(* Logix 5000 project; controller DispersionPlc vendor 1 type 14 code 108 rev 34.11; software revision 34.01; part 2 of 22 *)
(* tags used below, declared in another part *)
   TO_ALARM_MSG_DINT : DINT;

ADD_ON_INSTRUCTION AStd_VFD_AOI   (* revision 1.0 *)
VAR_IN_OUT
   VFD : AStd_VFD; {required}
END_VAR
VAR_INPUT
   Running_I : BOOL; {required}
   SpeedFdbk_I : REAL; {required}
   Disconnect_I : BOOL; {required}
   DriveFault_I : BOOL; {required}
END_VAR
VAR_OUTPUT
   Start_O : BOOL; {access Read Only, required}
   Stop_O : BOOL; {access Read Only, required}
   DirectionFWD_O : BOOL; {access Read Only, required}
   DirectionREV_O : BOOL; {required}
   SpeedCmd_O : REAL; {access Read Only, required}
   ClearFault_O : BOOL; {access Read Only, required}
   AutoS : BOOL; {access Read Only, visible}
   RunS : BOOL; {access Read Only, visible}
   ReverseS : BOOL; {access Read Only, visible}
   AlmS : BOOL; {access Read Only, visible}
END_VAR
VAR_INPUT
   cfgHasRunFdbk : BOOL := 1; {visible}
   cfgHasSpeedFdbk : BOOL := 1; {visible}
   cfgHasDISC : BOOL; {visible}
   cfgRawMin : REAL; {required}
   cfgRawMax : REAL := 32767.0; {required}
   cfgEUMin : REAL; {required}
   cfgEUMax : REAL := 100.0; {required}
END_VAR
VAR
   RuntimeHourTimer : TIMER := (PRE := 3600000); {access None}
END_VAR

ROUTINE Logic   (* ladder *)
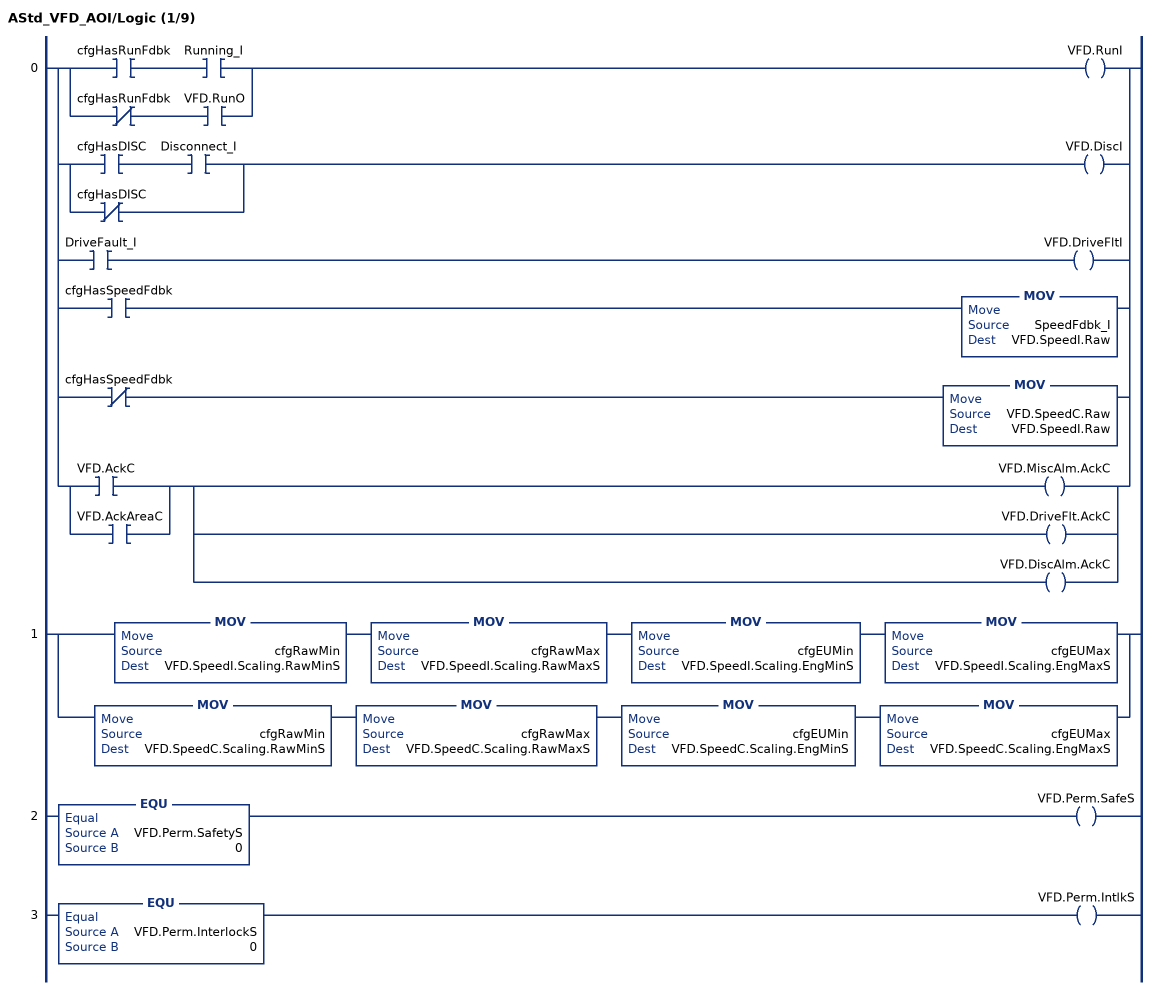
   0: [[XIC(cfgHasRunFdbk) XIC(Running_I) ,XIO(cfgHasRunFdbk) XIC(VFD.RunO) ] OTE(VFD.RunI) ,[XIC(cfgHasDISC) XIC(Disconnect_I) ,XIO(cfgHasDISC) ] OTE(VFD.DiscI) ,XIC(DriveFault_I) OTE(VFD.DriveFltI) ,[XIC(cfgHasSpeedFdbk) MOV(SpeedFdbk_I,VFD.SpeedI.Raw) ,XIO(cfgHasSpeedFdbk) MOV(VFD.SpeedC.Raw,VFD.SpeedI.Raw) ] ,[XIC(VFD.AckC) ,XIC(VFD.AckAreaC) ] [OTE(VFD.MiscAlm.AckC) ,OTE(VFD.DriveFlt.AckC) ,OTE(VFD.DiscAlm.AckC) ] ];
   1: [MOV(cfgRawMin,VFD.SpeedI.Scaling.RawMinS) MOV(cfgRawMax,VFD.SpeedI.Scaling.RawMaxS) MOV(cfgEUMin,VFD.SpeedI.Scaling.EngMinS) MOV(cfgEUMax,VFD.SpeedI.Scaling.EngMaxS) ,MOV(cfgRawMin,VFD.SpeedC.Scaling.RawMinS) MOV(cfgRawMax,VFD.SpeedC.Scaling.RawMaxS) MOV(cfgEUMin,VFD.SpeedC.Scaling.EngMinS) MOV(cfgEUMax,VFD.SpeedC.Scaling.EngMaxS) ];
   2: EQU(VFD.Perm.SafetyS,0)OTE(VFD.Perm.SafeS);
   3: EQU(VFD.Perm.InterlockS,0)OTE(VFD.Perm.IntlkS);
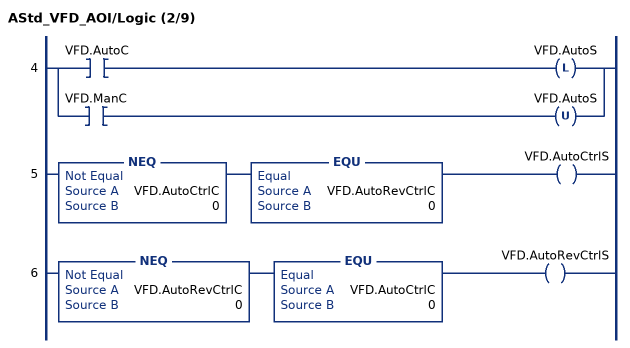
   4: [XIC(VFD.AutoC) OTL(VFD.AutoS) ,XIC(VFD.ManC) OTU(VFD.AutoS) ];
   5: NEQ(VFD.AutoCtrlC,0)EQU(VFD.AutoRevCtrlC,0)OTE(VFD.AutoCtrlS);
   6: NEQ(VFD.AutoRevCtrlC,0)EQU(VFD.AutoCtrlC,0)OTE(VFD.AutoRevCtrlS);
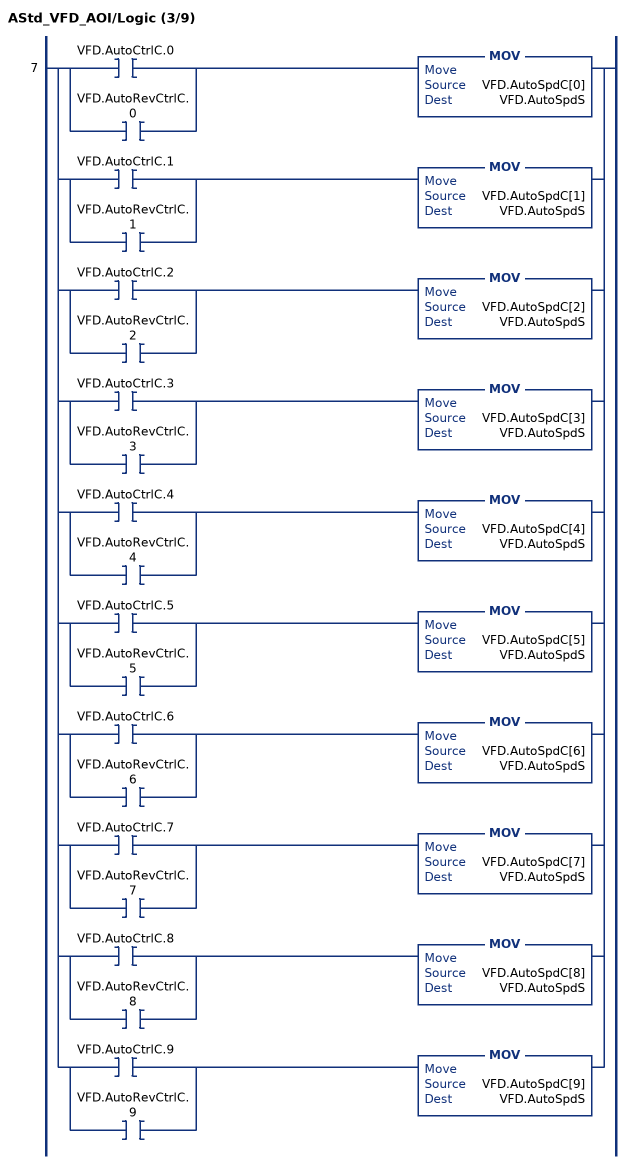
   7: [[XIC(VFD.AutoCtrlC.0) ,XIC(VFD.AutoRevCtrlC.0) ] MOV(VFD.AutoSpdC[0],VFD.AutoSpdS) ,[XIC(VFD.AutoCtrlC.1) ,XIC(VFD.AutoRevCtrlC.1) ] MOV(VFD.AutoSpdC[1],VFD.AutoSpdS) ,[XIC(VFD.AutoCtrlC.2) ,XIC(VFD.AutoRevCtrlC.2) ] MOV(VFD.AutoSpdC[2],VFD.AutoSpdS) ,[XIC(VFD.AutoCtrlC.3) ,XIC(VFD.AutoRevCtrlC.3) ] MOV(VFD.AutoSpdC[3],VFD.AutoSpdS) ,[XIC(VFD.AutoCtrlC.4) ,XIC(VFD.AutoRevCtrlC.4) ] MOV(VFD.AutoSpdC[4],VFD.AutoSpdS) ,[XIC(VFD.AutoCtrlC.5) ,XIC(VFD.AutoRevCtrlC.5) ] MOV(VFD.AutoSpdC[5],VFD.AutoSpdS) ,[XIC(VFD.AutoCtrlC.6) ,XIC(VFD.AutoRevCtrlC.6) ] MOV(VFD.AutoSpdC[6],VFD.AutoSpdS) ,[XIC(VFD.AutoCtrlC.7) ,XIC(VFD.AutoRevCtrlC.7) ] MOV(VFD.AutoSpdC[7],VFD.AutoSpdS) ,[XIC(VFD.AutoCtrlC.8) ,XIC(VFD.AutoRevCtrlC.8) ] MOV(VFD.AutoSpdC[8],VFD.AutoSpdS) ,[XIC(VFD.AutoCtrlC.9) ,XIC(VFD.AutoRevCtrlC.9) ] MOV(VFD.AutoSpdC[9],VFD.AutoSpdS) ];
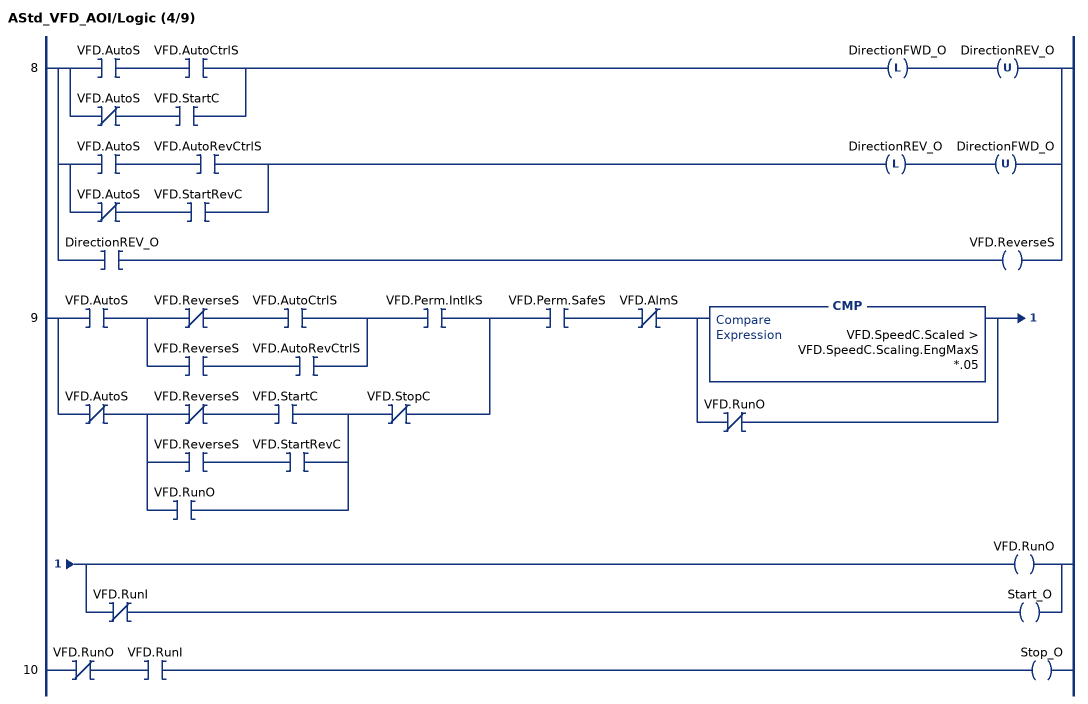
   8: [[XIC(VFD.AutoS) XIC(VFD.AutoCtrlS) ,XIO(VFD.AutoS) XIC(VFD.StartC) ] OTL(DirectionFWD_O) OTU(DirectionREV_O) ,[XIC(VFD.AutoS) XIC(VFD.AutoRevCtrlS) ,XIO(VFD.AutoS) XIC(VFD.StartRevC) ] OTL(DirectionREV_O) OTU(DirectionFWD_O) ,XIC(DirectionREV_O) OTE(VFD.ReverseS) ];
   9: [XIC(VFD.AutoS) [XIO(VFD.ReverseS) XIC(VFD.AutoCtrlS) ,XIC(VFD.ReverseS) XIC(VFD.AutoRevCtrlS) ] XIC(VFD.Perm.IntlkS) ,XIO(VFD.AutoS) [XIO(VFD.ReverseS) XIC(VFD.StartC) ,XIC(VFD.ReverseS) XIC(VFD.StartRevC) ,XIC(VFD.RunO) ] XIO(VFD.StopC) ]XIC(VFD.Perm.SafeS)XIO(VFD.AlmS)[CMP(VFD.SpeedC.Scaled > VFD.SpeedC.Scaling.EngMaxS *.05) ,XIO(VFD.RunO) ][OTE(VFD.RunO) ,XIO(VFD.RunI) OTE(Start_O) ];
   10: XIO(VFD.RunO)XIC(VFD.RunI)OTE(Stop_O);
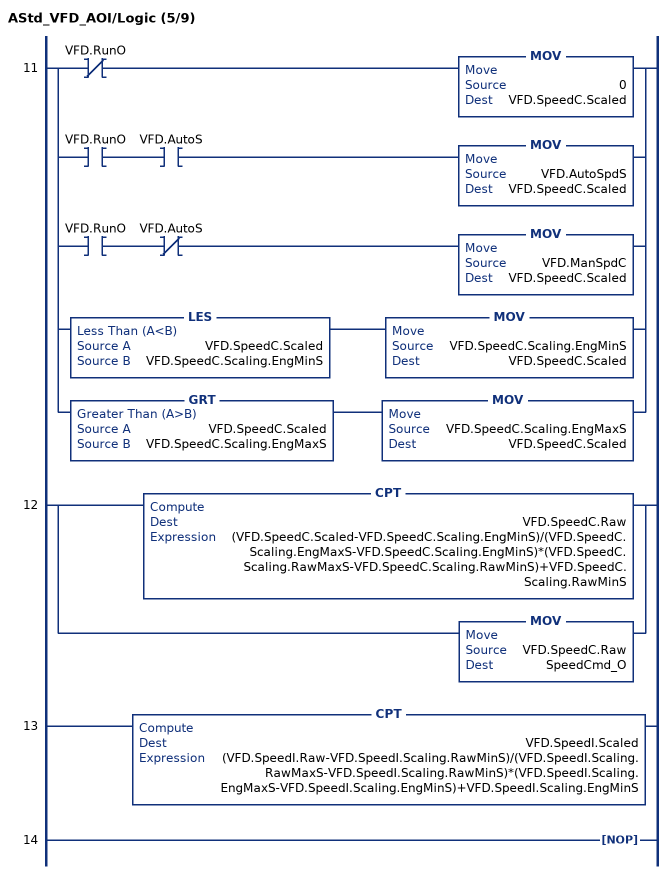
   11: [XIO(VFD.RunO) MOV(0,VFD.SpeedC.Scaled) ,XIC(VFD.RunO) XIC(VFD.AutoS) MOV(VFD.AutoSpdS,VFD.SpeedC.Scaled) ,XIC(VFD.RunO) XIO(VFD.AutoS) MOV(VFD.ManSpdC,VFD.SpeedC.Scaled) ,LES(VFD.SpeedC.Scaled,VFD.SpeedC.Scaling.EngMinS) MOV(VFD.SpeedC.Scaling.EngMinS,VFD.SpeedC.Scaled) ,GRT(VFD.SpeedC.Scaled,VFD.SpeedC.Scaling.EngMaxS) MOV(VFD.SpeedC.Scaling.EngMaxS,VFD.SpeedC.Scaled) ];
   12: [CPT(VFD.SpeedC.Raw,(VFD.SpeedC.Scaled-VFD.SpeedC.Scaling.EngMinS)/(VFD.SpeedC.Scaling.EngMaxS-VFD.SpeedC.Scaling.EngMinS)*(VFD.SpeedC.Scaling.RawMaxS-VFD.SpeedC.Scaling.RawMinS)+VFD.SpeedC.Scaling.RawMinS) ,MOV(VFD.SpeedC.Raw,SpeedCmd_O) ];
   13: CPT(VFD.SpeedI.Scaled,(VFD.SpeedI.Raw-VFD.SpeedI.Scaling.RawMinS)/(VFD.SpeedI.Scaling.RawMaxS-VFD.SpeedI.Scaling.RawMinS)*(VFD.SpeedI.Scaling.EngMaxS-VFD.SpeedI.Scaling.EngMinS)+VFD.SpeedI.Scaling.EngMinS);
   14: NOP();
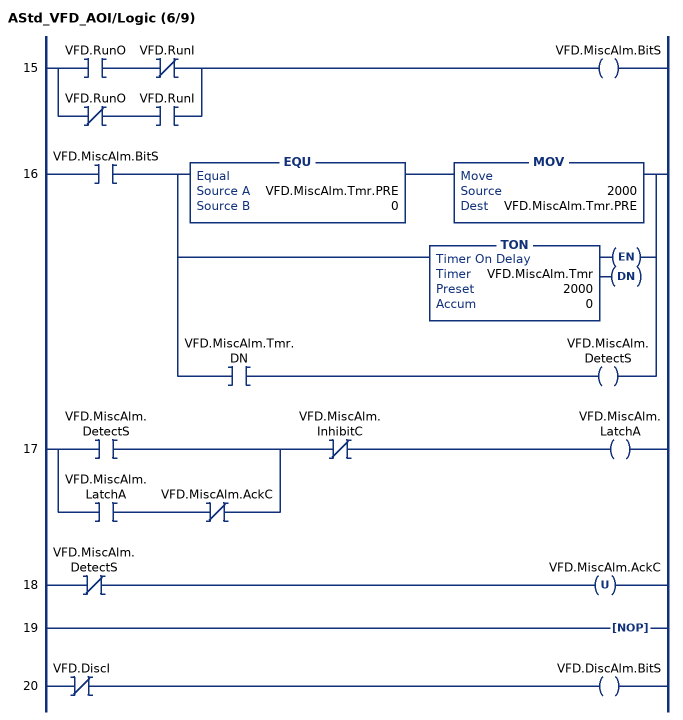
   15: [XIC(VFD.RunO) XIO(VFD.RunI) ,XIO(VFD.RunO) XIC(VFD.RunI) ]OTE(VFD.MiscAlm.BitS);
   16: XIC(VFD.MiscAlm.BitS)[EQU(VFD.MiscAlm.Tmr.PRE,0) MOV(2000,VFD.MiscAlm.Tmr.PRE) ,TON(VFD.MiscAlm.Tmr,2000,0) ,XIC(VFD.MiscAlm.Tmr.DN) OTE(VFD.MiscAlm.DetectS) ];
   17: [XIC(VFD.MiscAlm.DetectS) ,XIC(VFD.MiscAlm.LatchA) XIO(VFD.MiscAlm.AckC) ]XIO(VFD.MiscAlm.InhibitC)OTE(VFD.MiscAlm.LatchA);
   18: XIO(VFD.MiscAlm.DetectS)OTU(VFD.MiscAlm.AckC);
   19: NOP();
   20: XIO(VFD.DiscI)OTE(VFD.DiscAlm.BitS);
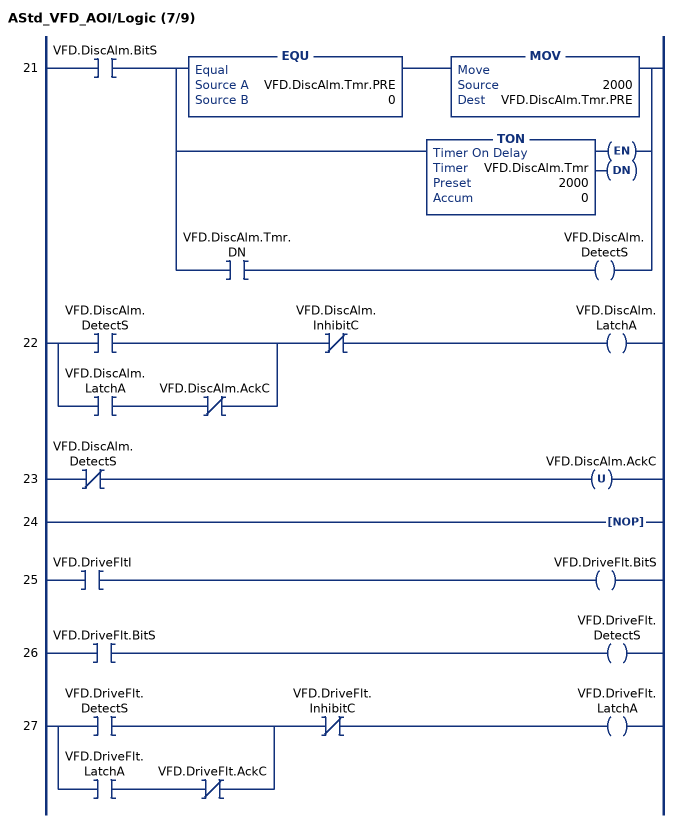
   21: XIC(VFD.DiscAlm.BitS)[EQU(VFD.DiscAlm.Tmr.PRE,0) MOV(2000,VFD.DiscAlm.Tmr.PRE) ,TON(VFD.DiscAlm.Tmr,2000,0) ,XIC(VFD.DiscAlm.Tmr.DN) OTE(VFD.DiscAlm.DetectS) ];
   22: [XIC(VFD.DiscAlm.DetectS) ,XIC(VFD.DiscAlm.LatchA) XIO(VFD.DiscAlm.AckC) ]XIO(VFD.DiscAlm.InhibitC)OTE(VFD.DiscAlm.LatchA);
   23: XIO(VFD.DiscAlm.DetectS)OTU(VFD.DiscAlm.AckC);
   24: NOP();
   25: XIC(VFD.DriveFltI)OTE(VFD.DriveFlt.BitS);
   26: XIC(VFD.DriveFlt.BitS)OTE(VFD.DriveFlt.DetectS);
   27: [XIC(VFD.DriveFlt.DetectS) ,XIC(VFD.DriveFlt.LatchA) XIO(VFD.DriveFlt.AckC) ]XIO(VFD.DriveFlt.InhibitC)OTE(VFD.DriveFlt.LatchA);
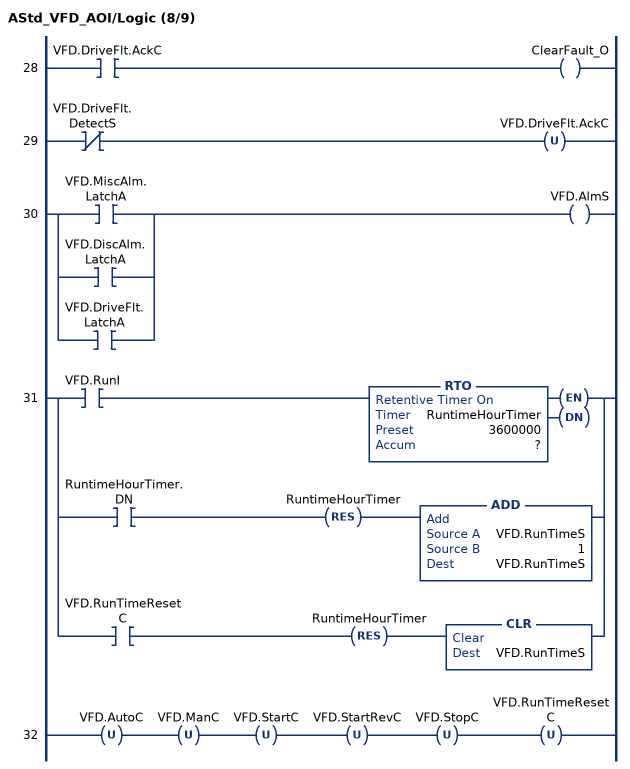
   28: XIC(VFD.DriveFlt.AckC)OTE(ClearFault_O);
   29: XIO(VFD.DriveFlt.DetectS)OTU(VFD.DriveFlt.AckC);
   30: [XIC(VFD.MiscAlm.LatchA) ,XIC(VFD.DiscAlm.LatchA) ,XIC(VFD.DriveFlt.LatchA) ]OTE(VFD.AlmS);
   31: [XIC(VFD.RunI) RTO(RuntimeHourTimer,?,?) ,XIC(RuntimeHourTimer.DN) RES(RuntimeHourTimer) ADD(VFD.RunTimeS,1,VFD.RunTimeS) ,XIC(VFD.RunTimeResetC) RES(RuntimeHourTimer) CLR(VFD.RunTimeS) ];
   32: OTU(VFD.AutoC)OTU(VFD.ManC)OTU(VFD.StartC)OTU(VFD.StartRevC)OTU(VFD.StopC)OTU(VFD.RunTimeResetC);
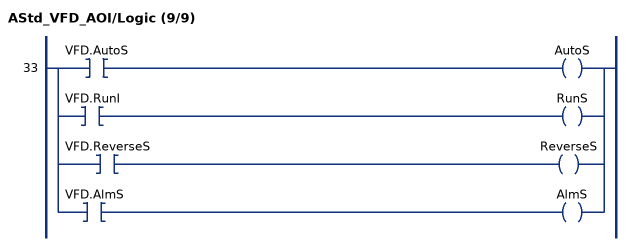
   33: [XIC(VFD.AutoS) OTE(AutoS) ,XIC(VFD.RunI) OTE(RunS) ,XIC(VFD.ReverseS) OTE(ReverseS) ,XIC(VFD.AlmS) OTE(AlmS) ];
END_ROUTINE
END_ADD_ON_INSTRUCTION

ADD_ON_INSTRUCTION AStd_VlVModulating_AOI   (* revision 1.0, vendor Avanceon *)
VAR_IN_OUT
   Valve : AStd_VlvModulating; {required}
END_VAR
VAR_INPUT
   cfgEUMin : REAL; {required}
   cfgEUMax : REAL := 100.0; {required}
   cfgRawMin : REAL := 4000.0; {required}
   cfgRawMax : REAL := 20000.0; {required}
END_VAR
VAR_OUTPUT
   OutputRaw_O : REAL; {required}
   AutoS : BOOL; {access Read Only, visible}
   OpenS : BOOL; {access Read Only, visible}
END_VAR
VAR
   ValveOpenRequest : BOOL; {access None}
END_VAR

ROUTINE Logic   (* ladder *)
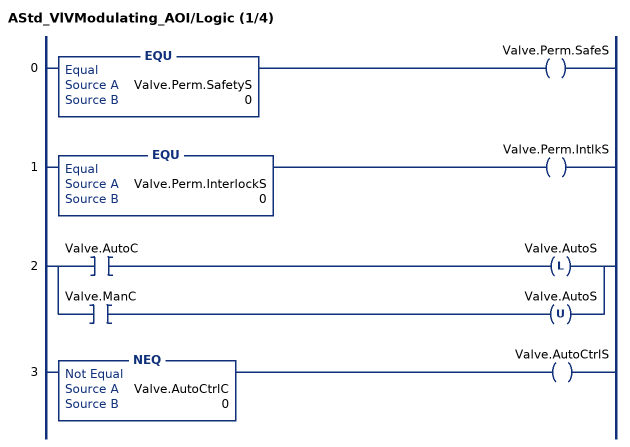
   0: EQU(Valve.Perm.SafetyS,0)OTE(Valve.Perm.SafeS);
   1: EQU(Valve.Perm.InterlockS,0)OTE(Valve.Perm.IntlkS);
   2: [XIC(Valve.AutoC) OTL(Valve.AutoS) ,XIC(Valve.ManC) OTU(Valve.AutoS) ];
   3: NEQ(Valve.AutoCtrlC,0)OTE(Valve.AutoCtrlS);
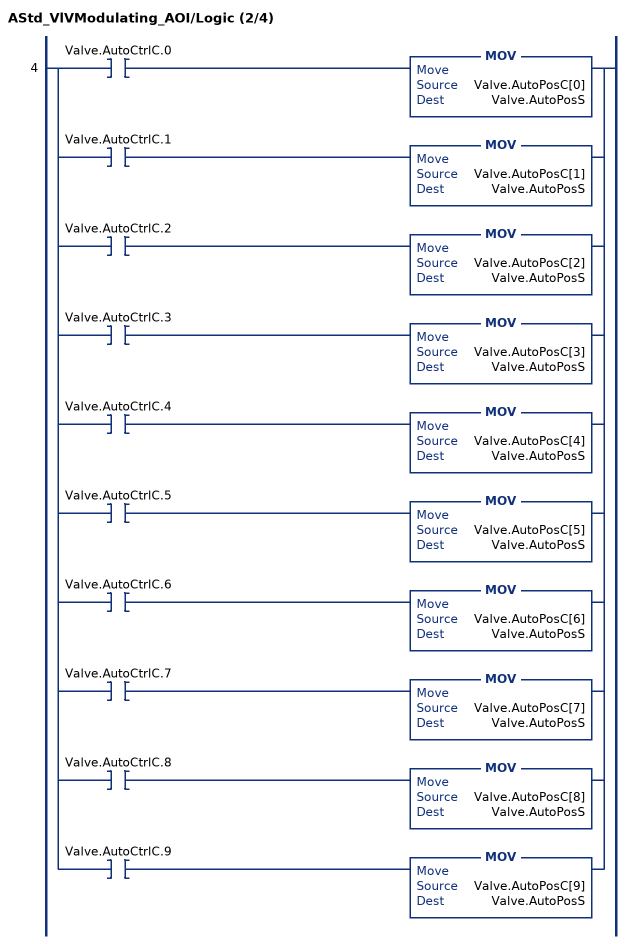
   4: [XIC(Valve.AutoCtrlC.0) MOV(Valve.AutoPosC[0],Valve.AutoPosS) ,XIC(Valve.AutoCtrlC.1) MOV(Valve.AutoPosC[1],Valve.AutoPosS) ,XIC(Valve.AutoCtrlC.2) MOV(Valve.AutoPosC[2],Valve.AutoPosS) ,XIC(Valve.AutoCtrlC.3) MOV(Valve.AutoPosC[3],Valve.AutoPosS) ,XIC(Valve.AutoCtrlC.4) MOV(Valve.AutoPosC[4],Valve.AutoPosS) ,XIC(Valve.AutoCtrlC.5) MOV(Valve.AutoPosC[5],Valve.AutoPosS) ,XIC(Valve.AutoCtrlC.6) MOV(Valve.AutoPosC[6],Valve.AutoPosS) ,XIC(Valve.AutoCtrlC.7) MOV(Valve.AutoPosC[7],Valve.AutoPosS) ,XIC(Valve.AutoCtrlC.8) MOV(Valve.AutoPosC[8],Valve.AutoPosS) ,XIC(Valve.AutoCtrlC.9) MOV(Valve.AutoPosC[9],Valve.AutoPosS) ];
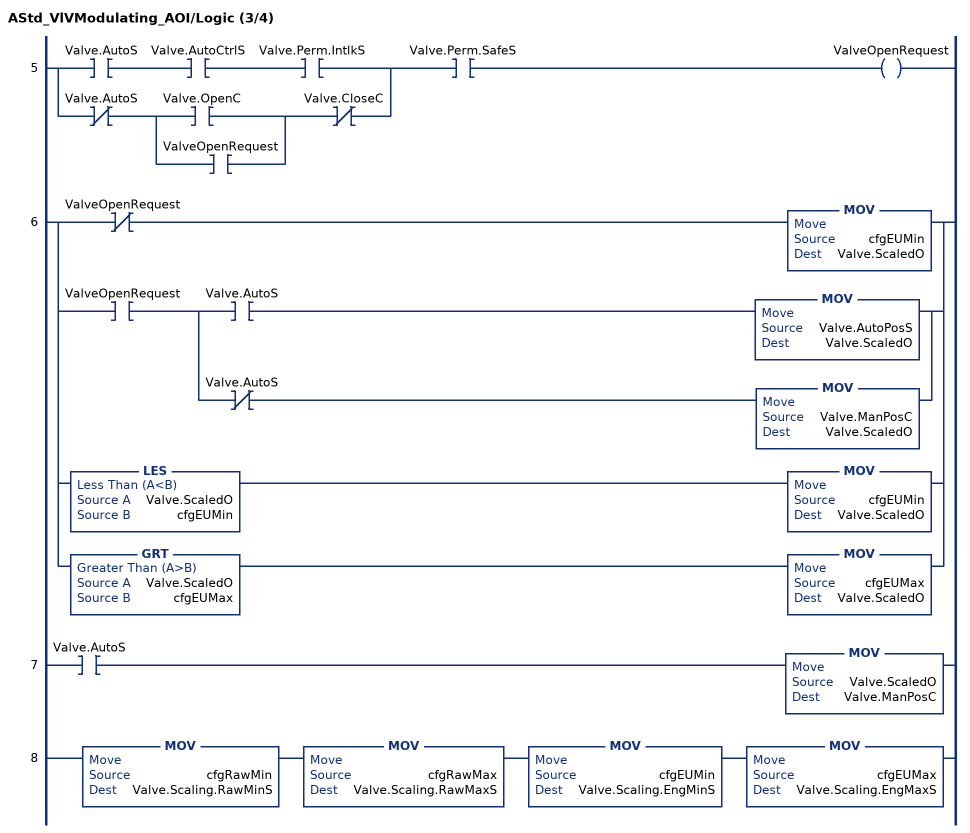
   5: [XIC(Valve.AutoS) XIC(Valve.AutoCtrlS) XIC(Valve.Perm.IntlkS) ,XIO(Valve.AutoS) [XIC(Valve.OpenC) ,XIC(ValveOpenRequest) ] XIO(Valve.CloseC) ]XIC(Valve.Perm.SafeS)OTE(ValveOpenRequest);
   6: [XIO(ValveOpenRequest) MOV(cfgEUMin,Valve.ScaledO) ,XIC(ValveOpenRequest) [XIC(Valve.AutoS) MOV(Valve.AutoPosS,Valve.ScaledO) ,XIO(Valve.AutoS) MOV(Valve.ManPosC,Valve.ScaledO) ] ,LES(Valve.ScaledO,cfgEUMin) MOV(cfgEUMin,Valve.ScaledO) ,GRT(Valve.ScaledO,cfgEUMax) MOV(cfgEUMax,Valve.ScaledO) ];
   7: XIC(Valve.AutoS)MOV(Valve.ScaledO,Valve.ManPosC);
   8: MOV(cfgRawMin,Valve.Scaling.RawMinS)MOV(cfgRawMax,Valve.Scaling.RawMaxS)MOV(cfgEUMin,Valve.Scaling.EngMinS)MOV(cfgEUMax,Valve.Scaling.EngMaxS);
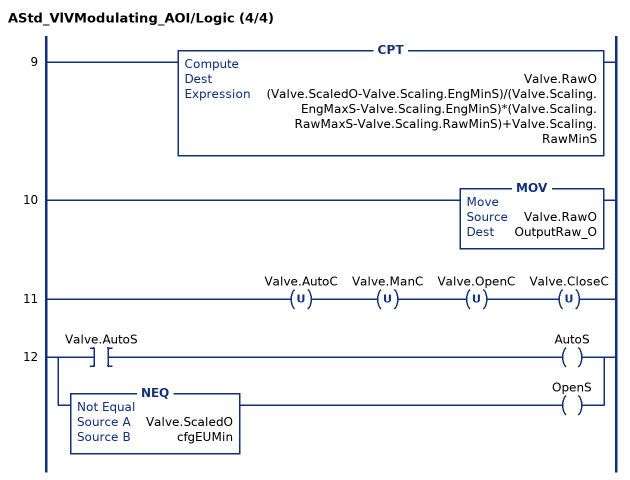
   9: CPT(Valve.RawO,(Valve.ScaledO-Valve.Scaling.EngMinS)/(Valve.Scaling.EngMaxS-Valve.Scaling.EngMinS)*(Valve.Scaling.RawMaxS-Valve.Scaling.RawMinS)+Valve.Scaling.RawMinS);
   10: MOV(Valve.RawO,OutputRaw_O);
   11: OTU(Valve.AutoC)OTU(Valve.ManC)OTU(Valve.OpenC)OTU(Valve.CloseC);
   12: [XIC(Valve.AutoS) OTE(AutoS) ,NEQ(Valve.ScaledO,cfgEUMin) OTE(OpenS) ];
END_ROUTINE
END_ADD_ON_INSTRUCTION

ADD_ON_INSTRUCTION AStd_VlvOC_AOI   (* revision 1.0, vendor Avanceon *)
VAR_IN_OUT
   Valve : AStd_VlvOC; {required}
END_VAR
VAR_OUTPUT
   AutoS : BOOL; {access Read Only, visible}
   OpenS : BOOL; {access Read Only, visible}
   AlmS : BOOL; {access Read Only, visible}
END_VAR
VAR_INPUT
   Open_I : BOOL; {required}
   Closed_I : BOOL; {required}
END_VAR
VAR_OUTPUT
   Open_O : BOOL; {required}
   Close_O : BOOL; {required}
END_VAR
VAR_INPUT
   cfgFailOpen : BOOL; {access None, visible}
   cfgHasZSO : BOOL := 1; {access None, visible}
   cfgHasZSC : BOOL; {access None, visible}
END_VAR
VAR
   ONS : SINT; {access None}
END_VAR

ROUTINE Logic   (* ladder *)
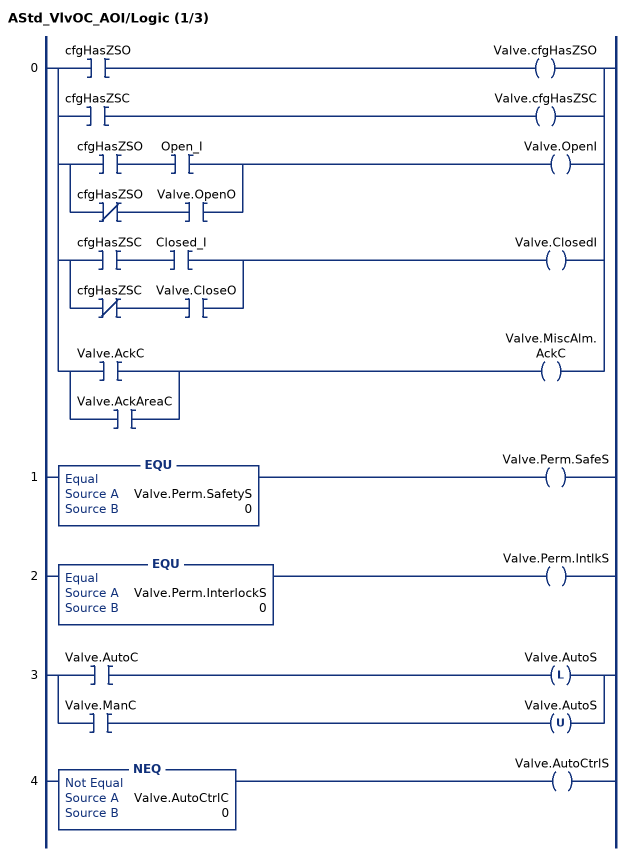
   0: [XIC(cfgHasZSO) OTE(Valve.cfgHasZSO) ,XIC(cfgHasZSC) OTE(Valve.cfgHasZSC) ,[XIC(cfgHasZSO) XIC(Open_I) ,XIO(cfgHasZSO) XIC(Valve.OpenO) ] OTE(Valve.OpenI) ,[XIC(cfgHasZSC) XIC(Closed_I) ,XIO(cfgHasZSC) XIC(Valve.CloseO) ] OTE(Valve.ClosedI) ,[XIC(Valve.AckC) ,XIC(Valve.AckAreaC) ] OTE(Valve.MiscAlm.AckC) ];
   1: EQU(Valve.Perm.SafetyS,0)OTE(Valve.Perm.SafeS);
   2: EQU(Valve.Perm.InterlockS,0)OTE(Valve.Perm.IntlkS);
   3: [XIC(Valve.AutoC) OTL(Valve.AutoS) ,XIC(Valve.ManC) OTU(Valve.AutoS) ];
   4: NEQ(Valve.AutoCtrlC,0)OTE(Valve.AutoCtrlS);
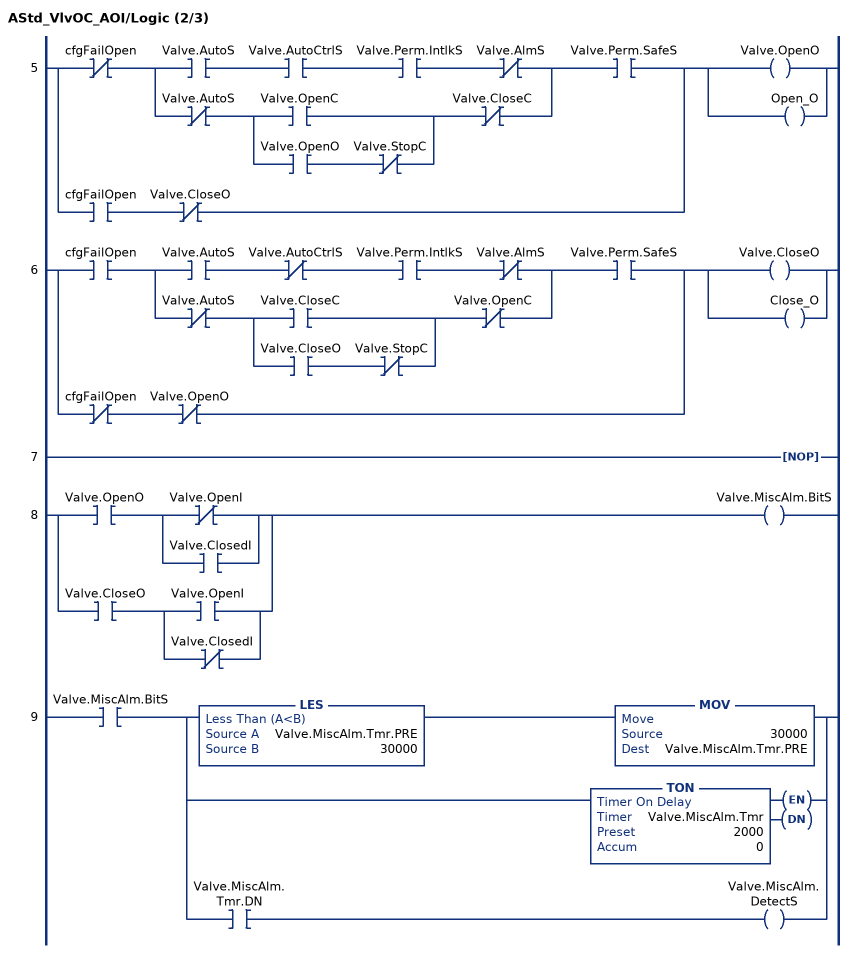
   5: [XIO(cfgFailOpen) [XIC(Valve.AutoS) XIC(Valve.AutoCtrlS) XIC(Valve.Perm.IntlkS) XIO(Valve.AlmS) ,XIO(Valve.AutoS) [XIC(Valve.OpenC) ,XIC(Valve.OpenO) XIO(Valve.StopC) ] XIO(Valve.CloseC) ] XIC(Valve.Perm.SafeS) ,XIC(cfgFailOpen) XIO(Valve.CloseO) ][OTE(Valve.OpenO) ,OTE(Open_O) ];
   6: [XIC(cfgFailOpen) [XIC(Valve.AutoS) XIO(Valve.AutoCtrlS) XIC(Valve.Perm.IntlkS) XIO(Valve.AlmS) ,XIO(Valve.AutoS) [XIC(Valve.CloseC) ,XIC(Valve.CloseO) XIO(Valve.StopC) ] XIO(Valve.OpenC) ] XIC(Valve.Perm.SafeS) ,XIO(cfgFailOpen) XIO(Valve.OpenO) ][OTE(Valve.CloseO) ,OTE(Close_O) ];
   7: NOP();
   8: [XIC(Valve.OpenO) [XIO(Valve.OpenI) ,XIC(Valve.ClosedI) ] ,XIC(Valve.CloseO) [XIC(Valve.OpenI) ,XIO(Valve.ClosedI) ] ]OTE(Valve.MiscAlm.BitS);
   9: XIC(Valve.MiscAlm.BitS)[LES(Valve.MiscAlm.Tmr.PRE,30000) MOV(30000,Valve.MiscAlm.Tmr.PRE) ,TON(Valve.MiscAlm.Tmr,2000,0) ,XIC(Valve.MiscAlm.Tmr.DN) OTE(Valve.MiscAlm.DetectS) ];
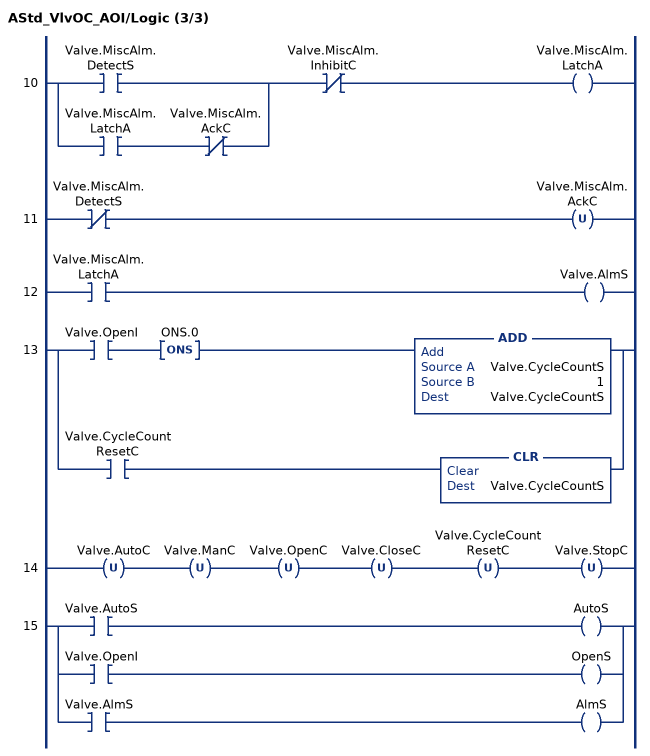
   10: [XIC(Valve.MiscAlm.DetectS) ,XIC(Valve.MiscAlm.LatchA) XIO(Valve.MiscAlm.AckC) ]XIO(Valve.MiscAlm.InhibitC)OTE(Valve.MiscAlm.LatchA);
   11: XIO(Valve.MiscAlm.DetectS)OTU(Valve.MiscAlm.AckC);
   12: XIC(Valve.MiscAlm.LatchA)OTE(Valve.AlmS);
   13: [XIC(Valve.OpenI) ONS(ONS.0) ADD(Valve.CycleCountS,1,Valve.CycleCountS) ,XIC(Valve.CycleCountResetC) CLR(Valve.CycleCountS) ];
   14: OTU(Valve.AutoC)OTU(Valve.ManC)OTU(Valve.OpenC)OTU(Valve.CloseC)OTU(Valve.CycleCountResetC)OTU(Valve.StopC);
   15: [XIC(Valve.AutoS) OTE(AutoS) ,XIC(Valve.OpenI) OTE(OpenS) ,XIC(Valve.AlmS) OTE(AlmS) ];
END_ROUTINE
END_ADD_ON_INSTRUCTION

VAR_GLOBAL   (* controller tags *)
   _bottom : REAL;
   _JISdebug : DINT := 2;
        .0   // Remapping
        .2   // Delete when probe is working
   _Placeholder : DINT := 1081857;
   _Placeholder_LS_4302_AI : REAL := 8.0;
   AFB : BOOL;
   AFI : BOOL;
   AG4302_LLP_Alarm : BOOL;
   AG4302_LLPower : TIMER := (PRE := 5000);
   AirMakeup : TIMER := (PRE := 2000);
   AirMakeup_BEAC : ALIAS FOR Local:1:O.Data[12].11;
   AirMakeup_BEACA : ALIAS FOR Local:1:O.Data[22].11;
   AMMONIUM_START_ATTEMP : BOOL;
   B4320_Amount_Per_Count : REAL;
   B4320_Charge_Remaining : REAL;
   B4320_Flow_Rate : REAL;
   B4320_Flow_Raw : DINT;
   B4320_Flow_Raw_Adjusted : REAL;
   B4320_Flow_Scale_Factor : REAL;
   B4320_HighHighLevel : BOOL;
   B4320_HighHighLevelMessage : BOOL;
   B4320_HighLevel : BOOL := 1;
   B4320_Last_Charge : DINT;
   B4320_LastTrasferredLb : REAL := 43900.0;
   B4320_Manual_Start : BOOL;
   B4320_Max_Flow : REAL;
   B4320_OkToRun : BOOL;
   B4320_Pump_Manual_Run : BOOL;
   B4320_Pump_Off : BOOL;
   B4320_Pump_Run : BOOL;
   B4320_PumpAutoCommand : BOOL;
   B4320_PumpManCommand : BOOL;
   B4320_PumpManStart : AOI_Toggle := (QNot := 1);
   B4320_Selected : BOOL;
   B4320_SelectPB : BOOL;
   B4320_Tank_Max_Lbs : REAL;
   B4320_Toggle : AOI_Toggle := (QNot := 1);
   B4320_Transfer : BOOL;
   B4320_transfer_amount : REAL;
   B4320_TransferDone : BOOL;
   B4320_TransferLimit : REAL := 44600.0;
   B4320_transferLimitMessage : BOOL;
   B4320_TransferSetpoint : REAL := 44000.0;
   B4320_TransferStarted : BOOL;
   B4320_TransferStartPB : BOOL;
   B4320_TransferStopPB : BOOL;
   B4320PumpTmr : TIMER;
   B4320SelectPB : BOOL;
   BarcodeBypassAcitve : BOOL;
   BarcodeBypassAcitvePB : BOOL;
   BarcodeForEditString : STRING := '01A0026';
   BarcodeIndex : DINT := 7;
   BarcodeIndex_Hold : DINT := 7;
   BarCodeReadHeartbeat : INT := 9751;
   BarcodeScan0NotOKDelay : TIMER := (PRE := 250);
   BarcodeScan1NotOKDelay : TIMER := (PRE := 250);
   BarcodeScan2NotOKDelay : TIMER := (PRE := 250);
   BarcodeScanBypass : BOOL := 1;
   BarcodeScanNotOK : INT;
   BarcodeScanOK : INT;
   BarcodeScanRequest : BOOL[32];
   BarcodeScanRequestPB : INT;
   BarcodeScanSequence : INT;
   bb : BOOL;
   BBVV : BOOL;
   BL_4310_AUX : ALIAS FOR Local:1:I.Data[1].2;
   BL_4310_RUN : ALIAS FOR Local:1:O.Data[0].2;
   BLANK64 : Stp64;
   BlankStrg : STRING;
   block_bit1 : BOOL := 1;
   block_bit2 : BOOL;
   bogus : BOOL;
   bogus_bit : BOOL;
   Both_Running : BOOL := 1;
   Both_Running_Timer : TIMER := (PRE := 3000, ACC := 3001, EN := 1, DN := 1);
   BUFENCTU : COUNTER := (PRE := 10000, ACC := 106);
   Bulk_Tank_T52_Level_Lamp : ALIAS FOR Local:1:O.Data[12].3;
   Bulk_Tank_T52_Level_LampA : ALIAS FOR Local:1:O.Data[12].3;
   Bulk_Tank_T52_Level_LampB : ALIAS FOR Local:1:O.Data[22].3;
   Bulk_Tank_T53_Level_Lamp : ALIAS FOR Local:1:O.Data[12].4;
   Bulk_Tank_T53_Level_LampA : ALIAS FOR Local:1:O.Data[22].4;
   bypass_bit : BOOL := 1;
   Capture_Delay : TIMER := (PRE := 3000);
   Capture_Delay_1 : TIMER := (PRE := 3000);
   Capture_Destination : DINT := 1;
   Capture_Destination_1 : DINT := 1;
   Capture_ONS : BOOL;
   Capture_ONS1 : BOOL;
   Capture_ONS_2 : BOOL;
   Capture_ONS_3 : BOOL;
   Capture_Selected : BOOL := 1;
   Capture_Selected_1 : BOOL;
   Cat_Destination_K400 : BOOL := 1;
   Cat_Destination_K400_ONS : BOOL;
   Cat_Destination_K400_PB : BOOL;
   Cat_Destination_T4301 : BOOL;
   Cat_Destination_T4301_ONS : BOOL;
   Cat_Destination_T4301_PB : BOOL;
   Cat_Destination_T4302 : BOOL;
   Cat_Destination_T4302_ONS : BOOL;
   Cat_Destination_T4302_PB : BOOL;
   Cat_Isolation_T430X_Timer : TIMER;
   Cat_Isolation_Valve_Timer : TIMER := (PRE := 120000);
   Cat_Man_ONS : BOOL;
   Cat_Pump_manual : BOOL;
   Cat_Purge_Transfer_K400 : Seq64 := (Sq.Step[0] := 1);
   Cat_Purge_Transfer_T430X : Seq64 := (Sq.Step[0] := 1);
   Cat_Recirc_Transfer_K400 : Seq64 := (Val := 6, Sq.Step[6] := 1);
   Cat_Recirc_Transfer_T430X : Seq64 := (Val := 1, Sq.Step[0] := 1);
   Cat_Scale_Factor : REAL := 0.0018;
   cat_start_dispencse : BOOL := 1;
   Cat_Tank_Destination : DINT := 1;
   cat_target_weight_bypass : BOOL;
   Cat_Zero : REAL := 4.03636;
   Catalyst_Destination : DINT;
   catalyst_MaxFeedRate : REAL := 3.4;
   CATALYST_RESET : BOOL;
   CatalystTimers_11_HMI : REAL := 7.01;
   CATFLOW : TIMER := (PRE := 500);
   CE_4301 : REAL := 0.17498249;
   ce_4301_High : REAL := 5.0;
   ce_4301_Low : REAL := -3.0;
   ce_4301_Max : REAL;
   CE_4301_OffSet : REAL := 4000.0;
   CE_4301_Sf : REAL := 0.0049995;
   CE_4302 : REAL := 0.129987;
   ce_4302_High : REAL := 15.0;
   CE_4302_Low : REAL := -3.0;
   CE_4302_OffSet : REAL := 4000.0;
   CE_4302_Sf : REAL := 0.0049995;
   Circulation_Timer_Continue : BOOL;
   constant : REAL := 10.0;
   constant1 : DINT := 1;
   Control_Rm_tags : DINT;
   Cool_Setpoint_4301 : DINT := 85;
   Cool_Setpoint_4302 : DINT := 180;
   Cool_SP : REAL := 15.0;
   Cool_SP2 : REAL := 17.5;
   Cool_SP3 : REAL := 20.0;
   Cool_SP4 : REAL := 100.0;
   CountTmr : TIMER := (PRE := 200);
   CR : STRING := '$0D';
   CRADT : ALIAS FOR Local:5:O.Data.7;
   Current4302FQ : REAL := 53.641064;
   CurrentTrasferredLb : REAL;
   dan1 : DINT := 112;
   dan2 : REAL := 1200.0;
   dan3 : BOOL;
   dan4 : BOOL := 1;
   dan5 : BOOL;
   dan6 : BOOL;
   dan99 : BOOL;
   dantoggle1 : BOOL := 1;
   DATAFDUNLATCH : TIMER := (PRE := 2000);
   DATAUNCOUNT : COUNTER := (PRE := 20000, ACC := 2198);
   ddd : BOOL := 1;
   Debug : DINT := 3;
   Dev : REAL[10] := ([0] := 2.8410683, [1] := 3.3833313);
   DevAck : DINT;
   DevAlarms : DINT := 60;
   DeviationFactor : REAL := 0.03;
   DevTimer : TIMER[10] := ([0].PRE := 30000, [1].PRE := 30000);
   Disp_AlarmsResetting : BOOL;
   Disp_Alr_To_Sound_Horn : BOOL[128] := ([10] := 1, [13] := 1, [14] := 1, [19] := 1, [25] := 1, [27] := 1, [28] := 1, [38] := 1, [44] := 1, [46] := 1, [51] := 1, [54] := 1, [55] := 1, [66] := 1, [70] := 1, [71] := 1, [87] := 1, [88] := 1, [99] := 1, [111] := 1, [115] := 1, [121] := 1, [122] := 1);
   Disp_AlrResetIdx : DINT := 127;
   Disp_QuedAlarm : DINT := 108;
   DispAlarmResetBit : BOOL;
   Dispersion_from_Main : DINT := 1;
   Dispersion_from_Main2 : DINT := 8131435;
   Dispersion_from_Main2_DintToStringConv : STRING := '8131435';
   Dispersion_from_SIL2 : DINT := 1;
   Dispersion_from_SIL2_Analog : REAL[24] := ([0] := 86.51327, [1] := 66.32967, [2] := 90.0, [10] := 152.36926);
   Dispersion_to_Main : DINT := 1;
   Dispersion_to_Main2 : DINT;
   Dispersion_to_SIL2 : DINT := 32;
   Dispersion_to_SIL2_Analog : REAL[24] := ([0] := 90.0, [1] := 10.0, [2] := 45.0, [3] := 15901.0, [4] := 15801.0);
   Dispersion_to_SIL2_Analog_xxx : DINT;
   DispersionAlarmReset : BOOL;
   DispersionAlarms : BOOL[256] := ([2] := 1, [103] := 1, [108] := 1, [157] := 1, [159] := 1, [250] := 1);
   DispersionProductID : STRING[21] := ([0] := '8131428', [1] := '8131435', [2] := '8132028', [3] := '8211377', [4] := '8212241', [5] := 'IDLE', [6] := '7108441');
   DispersionProductID_BarcodeScan : STRING;
   DispersionProductID_ScanIndex : DINT := 8;
   DispersionProductID_ScanIndex_Storage : DINT;
   DispersionProductIDEntryStorage : STRING;
   DispersionProductIDKeyEntry : STRING := '7108441';
   DispersionProductIDKeyEntry1 : STRING;
   DispersionProductIDMatch : STRING;
   DPT_4301 : REAL;
   dpt_4301_High : REAL := 40000.0;
   DPT_4301_Holding : REAL := 3900.84;
   DPT_4301_OffSet : REAL := 4000.0;
   DPT_4301_Samples : DINT := 1000;
   DPT_4301_Sf : REAL := 3.41875;
   DPT_4302 : REAL;
   dpt_4302_High : REAL := 35000.0;
   DPT_4302_Holding : REAL := 3917.319;
   DPT_4302_OffSet : REAL := 4000.0;
   DPT_4302_Samples : DINT := 100;
   DPT_4302_Sf : REAL := 3.41875;
   DPT_4303 : REAL := 7949.331;
   DPT_4303_High : REAL := 16300.0;
   DPT_4303_Holding : REAL := 10860.054;
   DPT_4303_OffSet : REAL := 4000.0;
   DPT_4303_Samples : DINT := 100;
   DPT_4303_Sf : REAL := 1.02186;
   DPT_4303_Tare_Val : REAL;
   DPT_4320 : REAL := 33840.145;
   DPT_4320_FILL : REAL := 1489.0;
   DPT_4320_High : REAL := 48500.0;
   DPT_4320_Holding1 : REAL := 14397.525;
   DPT_4320_OffSet : REAL := 3904.0;
   DPT_4320_Raw : INT := 14392;
   DPT_4320_Sf : REAL := 3.083;
   DPT_4320_Sf_old : REAL := 3.466;
   DPT_4320rev1 : REAL;
   dpthighraw : REAL := 20837.0;
   dptlowraw : REAL := -32.0;
   Drum_Addition_K400 : Seq64 := (Sq.Step[0] := 1, AutoMode := 1);
   Drum_Addition_T430X : Seq64 := (Sq.Step[0] := 1);
   Drum_Addition_T430X_Timer : TIMER := (PRE := 30000);
   Drum_Addition_Timer : TIMER := (PRE := 120000);
   Drum_Transfer : BOOL;
   Drum_Transfer_Active : BOOL;
   Drum_Transfer_ONS : BOOL;
   Drum_Transfer_ONS_1 : BOOL;
   Dummy_Safety_1 : BOOL[32];
   DummyOutput : BOOL := 1; {access None}
   Emergency_Cool_4301 : BOOL;
   Emergency_Cool_4301_Reset : BOOL;
   Emergency_Cool_4302 : BOOL;
   Emergency_Cool_4302_Reset : BOOL;
   Enable_High_Alarm : BOOL := 1;
   Enable_HMI_PB_SV4303 : BOOL;
   Enable_Shortstop_Automation : BOOL;
   Enable_TO_Message : BOOL := 1;
   Estop : BOOL;
   Estop_Bulk : ALIAS FOR Local:1:I.Data[33].5;
   Estop_Bulk_Upper : ALIAS FOR Estop_Bulk;
   Estop_Disp : ALIAS FOR Local:3:I.Data.1;
   Estop_Inx : ALIAS FOR Local:3:I.Data.3;
   Estop_Mcc : ALIAS FOR Local:3:I.Data.2;
   EstopBulk_upper : ALIAS FOR Local:1:O.Data[27].15;
   Fault_Reset_High : REAL := 17.0;
   Faut_Reset_Low : REAL := 7.0;
   FC_4302_1 : AStd_PIDInterface := (AutoS := 1, SPC := 59.0, PGainC := 1.95, IGainC := 0.5, PGainS := 1.95, IGainS := 0.5, SPS := 59.0, PVS := -0.7625, Perm.IntlkS := 1, Perm.SafeS := 1);
   FC_4302_1_AOI : AStd_PIDInterface_AOI := (SP := 59.0, PV := -0.7625, cfgPVMaxEU := 200.0);
   FC_4302_1_PID : PID_ENHANCED := (PV := -0.7625, PVEUMax := 200.0, SPProg := 59.0, SPOper := 59.0, SPHLimit := 200.0, RatioProg := 1.0, RatioOper := 1.0, RatioHLimit := 1.0, RatioLLimit := 1.0, CVEUMax := 100.0, CVHLimit := 100.0, DependIndepend := 1, PGain := 1.95, IGain := 0.5, PVHHLimit := 200.0, PVHLimit := 199.0, PVLLimit := 1.0, DevHHLimit := 10.0, DevDeadband := 2.0, ProgProgReq := 1, ProgOverrideReq := 1, RTSTime := 1, SP := 59.0, SPPercent := 29.499998, PVPercent := -0.38125, E := 59.7625, EPercent := 29.881248, InitPrimary := 1, Ratio := 1.0, PVLAlarm := 1, PVLLAlarm := 1, ProgOper := 1, Override := 1, DeltaT := 0.1);
   FC_4305_xx : AStd_PIDInterface := (AutoS := 1, SPC := 59.0, PGainC := 2.0, IGainC := 0.5, PGainS := 2.0, IGainS := 0.5, SPS := 59.0, PVS := -1.5, Perm.IntlkS := 1, Perm.SafeS := 1);
   FC_4305_xx_AOI : AStd_PIDInterface_AOI := (SP := 59.0, PV := -1.275, cfgPVMaxEU := 400.0);
   FC_4305_xx_PID : PID_ENHANCED := (PV := -1.35, PVEUMax := 400.0, SPProg := 59.0, SPOper := 59.0, SPHLimit := 400.0, RatioProg := 1.0, RatioOper := 1.0, RatioHLimit := 1.0, RatioLLimit := 1.0, CVEUMax := 100.0, CVHLimit := 100.0, CVLLimit := 25.0, DependIndepend := 1, PGain := 2.0, IGain := 0.5, PVHHLimit := 400.0, PVHLimit := 399.9, PVLLimit := 0.01, PVLLLimit := 0.01, DevHHLimit := 5.0, ProgProgReq := 1, ProgOverrideReq := 1, RTSTime := 1, CVLAlarm := 1, SP := 59.0, SPPercent := 14.749999, PVPercent := -0.33124998, E := 60.325, EPercent := 15.081249, InitPrimary := 1, WindupLOut := 1, Ratio := 1.0, PVLAlarm := 1, PVLLAlarm := 1, ProgOper := 1, Override := 1, DeltaT := 0.1);
   FCV_4302_1 : AStd_VlvModulating := (AutoC := 1, AutoS := 1, Perm.IntlkS := 1, Perm.SafeS := 1, AutoPosC[3] := 100.0, AutoPosC[4] := 100.0, AutoPosS := 100.0, Scaling.RawMaxS := 10000.0, Scaling.EngMaxS := 100.0);
   FCV_4302_1_AOI : AStd_VlVModulating_AOI := (cfgEUMax := 100.0, cfgRawMax := 10000.0, AutoS := 1);
   FCV_4305 : ALIAS FOR Local:13:O.Ch0Data;
   FCV_4305_Math : DINT := 4050;
   FCV_4305_OffSet : REAL := 4000.0;
   FCV_4305_Sf : REAL := 1.0;
   FCV_4305_SP : REAL := 4640.0;
   FCV_SCREEN_VALUE : REAL := 29.0;
   FE_4301_CW : REAL;
   FE_4301_CW_OffSet : REAL := 4000.0;
   FE_4301_CW_Sf : REAL := 1.0;
   FE_4301_RO : REAL;
   FE_4302_CW : REAL;
   FE_4302_CW_OffSet : REAL := 4000.0;
   FE_4302_CW_Sf : REAL := 1.0;
   FE_4302_RO : REAL;
   FE_4302_RO_OffSet : REAL := 4000.0;
   FE_4302_RO_Sf : REAL := 1.0;
   FE_4303 : REAL := 21.884998;
   FE_4303_AOI : Analog_Scale := (Analog_In := 8340.0, Offset_In := -4000.0, Analog_Min_In := 4000.0, Analog_Max_In := 20000.0, Analog_Max_Out := 80.0, Analog_Out := 21.699999);
   FE_4303_AVERAGE : MOVING_AVERAGE := (In := 21.74, SampleEnable := 1, NumberOfSamples := 50, Out := 21.864698);
   FE_4303_Corrected : REAL := 21.8821;
   FE_4303_Correction_Sf : REAL := 1.0;
   FE_4303_Low : REAL := 1.0;
   FE_4303_OffSet : REAL := -4000.0;
   FE_4303_OffSet_Out : REAL;
   FE_4303_Out : REAL := 22.15;
   FE_4303_Sf : REAL := 0.0031135;
   FE_4303_STORAGE : REAL[1000] := ([0] := 22.0, [1] := 21.725, [2] := 21.705, [3] := 22.095, [4] := 21.855, [5] := 22.119999, [6] := 21.71, [7] := 22.185, [8] := 22.07, [9] := 21.984999, [10] := 21.875, [11] := 21.72, [12] := 22.175, [13] := 21.689999, [14] := 21.805, [15] := 21.935, [16] := 21.984999, [17] := 21.77, [18] := 21.675, [19] := 22.16, [20] := 21.789999, [21] := 21.975, [22] := 21.789999, [23] := 22.119999, [24] := 22.15, [25] := 21.71, [26] := 22.07, [27] := 21.81, [28] := 22.119999, [29] := 21.685, [30] := 21.66, [31] := 22.025, [32] := 21.755, [33] := 21.88, [34] := 21.605, [35] := 21.975, [36] := 21.5, [37] := 21.56, [38] := 21.765, [39] := 21.845, [40] := 22.0, [41] := 21.585, [42] := 22.015, [43] := 21.855, [44] := 21.895, [45] := 21.615, [46] := 21.615, [47] := 22.029999, [48] := 21.734999, [49] := 21.89, [50] := 21.734999, [51] := 22.085, [52] := 21.654999, [53] := 21.689999, [54] := 22.05, [55] := 21.869999, [56] := 22.085, [57] := 21.81, [58] := 22.215, [59] := 22.14,
        [60] := 21.875, [61] := 21.93, [62] := 21.76, [63] := 22.154999, [64] := 21.67, [65] := 21.785, [66] := 21.695, [67] := 22.115, [68] := 21.67, [69] := 21.81, [70] := 21.755, [71] := 22.055, [72] := 22.09, [73] := 21.625, [74] := 21.91, [75] := 21.734999, [76] := 22.039999, [77] := 21.625, [78] := 21.705, [79] := 21.93, [80] := 21.865, [81] := 21.664999, [82] := 21.59, [83] := 22.045, [84] := 21.66, [85] := 21.82, [86] := 21.73, [87] := 21.975, [88] := 22.0, [89] := 21.75, [90] := 21.865, [91] := 21.75, [92] := 22.13, [93] := 21.699999, [94] := 21.765, [95] := 21.984999, [96] := 22.029999, [97] := 21.814999, [98] := 21.71, [99] := 22.185, [100] := 21.75, [101] := 21.91, [102] := 21.824999, [103] := 22.21, [104] := 22.185, [105] := 21.855, [106] := 22.06, [107] := 21.855, [108] := 22.14, [109] := 21.699999, [110] := 22.164999, [111] := 22.064999, [112] := 21.83, [113] := 21.91, [114] := 21.73, [115] := 22.105, [116] := 22.029999, [117] := 21.734999, [118] := 21.84, [119] := 21.89,
        [120] := 22.045, [121] := 21.63, [122] := 21.895, [123] := 21.615, [124] := 22.01, [125] := 21.57, [126] := 21.67, [127] := 22.005, [128] := 21.84, [129] := 21.82, [130] := 21.63, [131] := 22.0, [132] := 21.67, [133] := 21.83, [134] := 21.564999, [135] := 22.015, [136] := 22.005, [137] := 21.685, [138] := 21.895, [139] := 21.73, [140] := 22.055, [141] := 21.664999, [142] := 21.76, [143] := 21.99, [144] := 21.925, [145] := 22.135, [146] := 21.68, [147] := 22.039999, [148] := 21.814999, [149] := 22.095, [150] := 21.68, [151] := 22.15, [152] := 21.975, [153] := 21.9, [154] := 21.795, [155] := 21.675, [156] := 22.115, [157] := 21.71, [158] := 21.869999, [159] := 21.699999, [160] := 22.09, [161] := 21.635, [162] := 21.8, [163] := 21.914999, [164] := 21.984999, [165] := 22.135, [166] := 21.67, [167] := 21.984999, [168] := 21.755, [169] := 21.99, [170] := 21.59, [171] := 21.585, [172] := 21.84, [173] := 21.73, [174] := 21.675, [175] := 21.564999, [176] := 22.039999, [177] := 21.564999, [178] := 21.695, [179] := 21.869999,
        [180] := 21.885, [181] := 22.095, [182] := 21.66, [183] := 21.98, [184] := 21.72, [185] := 22.055, [186] := 21.63, [187] := 21.66, [188] := 21.91, [189] := 21.904999, [190] := 21.73, [191] := 21.65, [192] := 22.025, [193] := 21.885, [194] := 22.085, [195] := 21.734999, [196] := 22.215, [197] := 22.13, [198] := 21.904999, [199] := 21.85, [200] := 21.74, [201] := 22.199999, [202] := 21.72, [203] := 21.83, [204] := 21.9, [205] := 22.0, [206] := 21.689999, [207] := 21.675, [208] := 22.064999, [209] := 21.765, [210] := 22.074999, [211] := 21.615, [212] := 22.1, [213] := 22.01, [214] := 21.904999, [215] := 21.84, [216] := 22.07, [217] := 22.164999, [218] := 21.76, [219] := 21.914999, [220] := 21.699999, [221] := 22.145, [222] := 21.734999, [223] := 21.96, [224] := 21.605, [225] := 22.035, [226] := 21.855, [227] := 21.965, [228] := 21.515, [229] := 21.949999, [230] := 21.814999, [231] := 21.895, [232] := 22.015, [233] := 21.55, [234] := 22.029999, [235] := 21.789999, [236] := 22.01, [237] := 21.71, [238] := 22.145, [239] := 22.06,
        [240] := 21.84, [241] := 21.88, [242] := 21.715, [243] := 22.085, [244] := 21.609999, [245] := 22.08, [246] := 21.949999, [247] := 21.805, [248] := 21.984999, [249] := 21.64, [250] := 22.085, [251] := 21.779999, [252] := 21.939999, [253] := 21.77, [254] := 22.095, [255] := 22.16, [256] := 21.76, [257] := 21.994999, [258] := 21.82, [259] := 22.08, [260] := 21.699999, [261] := 22.154999, [262] := 22.09, [263] := 21.785, [264] := 21.92, [265] := 21.75, [266] := 22.074999, [267] := 21.775, [268] := 21.97, [269] := 21.744999, [270] := 22.08, [271] := 22.02, [272] := 21.685, [273] := 21.82, [274] := 21.625, [275] := 21.925, [276] := 21.484999, [277] := 21.955, [278] := 21.685, [279] := 21.875, [280] := 21.564999, [281] := 21.545, [282] := 21.895, [283] := 21.715, [284] := 21.904999, [285] := 21.55, [286] := 22.035, [287] := 21.975, [288] := 21.984999, [289] := 21.67, [290] := 21.65, [291] := 22.135, [292] := 22.0, [293] := 21.845, [294] := 21.76, [295] := 22.24, [296] := 21.949999, [297] := 22.1, [298] := 21.755, [299] := 22.18,
        [300] := 22.14, [301] := 21.77, [302] := 21.98, [303] := 21.76, [304] := 22.045, [305] := 21.65, [306] := 22.13, [307] := 22.09, [308] := 21.8, [309] := 22.039999, [310] := 21.64, [311] := 22.109999, [312] := 21.695, [313] := 21.845, [314] := 21.824999, [315] := 22.015, [316] := 22.135, [317] := 21.664999, [318] := 22.14, [319] := 22.01, [320] := 21.97, [321] := 21.84, [322] := 22.125, [323] := 22.164999, [324] := 21.744999, [325] := 21.98, [326] := 21.785, [327] := 22.1, [328] := 21.64, [329] := 21.71, [330] := 21.994999, [331] := 21.869999, [332] := 22.145, [333] := 21.705, [334] := 22.195, [335] := 22.13, [336] := 21.945, [337] := 21.96, [338] := 21.779999, [339] := 22.26, [340] := 21.82, [341] := 22.185, [342] := 21.805, [343] := 22.265, [344] := 21.814999, [345] := 21.939999, [346] := 21.865, [347] := 22.18, [348] := 22.215, [349] := 21.744999, [350] := 22.125, [351] := 21.949999, [352] := 22.039999, [353] := 21.71, [354] := 21.8, [355] := 22.06, [356] := 22.074999, [357] := 21.785, [358] := 21.685, [359] := 22.145,
        [360] := 21.715, [361] := 21.875, [362] := 21.82, [363] := 22.01, [364] := 22.1, [365] := 21.615, [366] := 22.05, [367] := 21.789999, [368] := 21.949999, [369] := 21.64, [370] := 21.609999, [371] := 21.965, [372] := 21.74, [373] := 21.789999, [374] := 21.574999, [375] := 22.035, [376] := 21.574999, [377] := 21.699999, [378] := 21.785, [379] := 21.869999, [380] := 22.025, [381] := 21.605, [382] := 22.035, [383] := 21.885, [384] := 21.92, [385] := 21.64, [386] := 22.085, [387] := 22.05, [388] := 21.74, [389] := 21.835, [390] := 21.734999, [391] := 22.205, [392] := 21.795, [393] := 21.97, [394] := 21.97, [395] := 22.135, [396] := 22.255, [397] := 21.775, [398] := 22.225, [399] := 21.859999, [400] := 22.15, [401] := 21.725, [402] := 22.185, [403] := 22.01, [404] := 21.945, [405] := 21.84, [406] := 21.689999, [407] := 22.15, [408] := 21.734999, [409] := 21.89, [410] := 21.744999, [411] := 22.119999, [412] := 22.115, [413] := 21.76, [414] := 21.869999, [415] := 21.685, [416] := 22.029999, [417] := 21.619999, [418] := 21.775, [419] := 21.734999,
        [420] := 21.955, [421] := 21.595, [422] := 21.74, [423] := 21.865, [424] := 22.005, [425] := 22.1, [426] := 21.615, [427] := 22.05, [428] := 21.779999, [429] := 21.975, [430] := 21.609999, [431] := 22.055, [432] := 21.81, [433] := 21.875, [434] := 21.675, [435] := 21.654999, [436] := 21.98, [437] := 21.85, [438] := 22.025, [439] := 21.71, [440] := 22.14, [441] := 22.115, [442] := 21.945, [443] := 21.77, [444] := 22.1, [445] := 22.14, [446] := 21.765, [447] := 21.96, [448] := 21.835, [449] := 22.119999, [450] := 21.695, [451] := 21.765, [452] := 21.91, [453] := 22.02, [454] := 22.15, [455] := 21.685, [456] := 22.154999, [457] := 21.93, [458] := 21.955, [459] := 21.75, [460] := 22.125, [461] := 21.994999, [462] := 21.85, [463] := 21.725, [464] := 21.63, [465] := 22.119999, [466] := 21.689999, [467] := 21.935, [468] := 21.744999, [469] := 22.074999, [470] := 22.14, [471] := 21.765, [472] := 21.96, [473] := 21.765, [474] := 22.07, [475] := 21.765, [476] := 21.93, [477] := 21.789999, [478] := 22.164999, [479] := 21.74,
        [480] := 21.895, [481] := 21.785, [482] := 22.17, [483] := 22.109999, [484] := 21.76, [485] := 21.75, [486] := 22.09, [487] := 22.115, [488] := 21.66, [489] := 21.685, [490] := 21.574999, [491] := 22.05, [492] := 21.625, [493] := 21.914999, [494] := 21.715, [495] := 22.08, [496] := 21.984999, [497] := 21.845, [498] := 21.785, [499] := 21.609999, [500] := 22.085, [501] := 21.65, [502] := 21.98, [503] := 21.699999, [504] := 22.029999, [505] := 21.585, [506] := 21.595, [507] := 21.97, [508] := 21.715, [509] := 21.965, [510] := 21.56, [511] := 22.01, [512] := 21.945, [513] := 21.755, [514] := 21.699999, [515] := 21.945, [516] := 22.06, [517] := 21.605, [518] := 22.0, [519] := 21.88, [520] := 22.085, [521] := 21.715, [522] := 21.75, [523] := 22.095, [524] := 21.925, [525] := 22.189999, [526] := 21.755, [527] := 22.225, [528] := 21.824999, [529] := 22.175, [530] := 21.715, [531] := 22.18, [532] := 22.039999, [533] := 21.824999, [534] := 21.83, [535] := 21.59, [536] := 22.05, [537] := 21.58, [538] := 21.805, [539] := 21.6,
        [540] := 22.025, [541] := 22.05, [542] := 21.775, [543] := 21.859999, [544] := 21.689999, [545] := 22.07, [546] := 21.67, [547] := 21.88, [548] := 21.68, [549] := 21.93, [550] := 21.5, [551] := 21.56, [552] := 21.835, [553] := 21.83, [554] := 21.99, [555] := 21.529999, [556] := 22.02, [557] := 21.93, [558] := 21.785, [559] := 21.755, [560] := 21.945, [561] := 22.039999, [562] := 21.585, [563] := 22.05, [564] := 21.945, [565] := 21.92, [566] := 21.789999, [567] := 21.67, [568] := 22.145, [569] := 21.779999, [570] := 21.945, [571] := 21.755, [572] := 22.145, [573] := 22.15, [574] := 21.845, [575] := 21.93, [576] := 21.765, [577] := 22.16, [578] := 21.725, [579] := 22.154999, [580] := 22.039999, [581] := 22.095, [582] := 21.81, [583] := 21.785, [584] := 22.189999, [585] := 21.869999, [586] := 21.8, [587] := 21.695, [588] := 22.16, [589] := 21.949999, [590] := 22.02, [591] := 21.805, [592] := 22.175, [593] := 22.205, [594] := 21.76, [595] := 22.085, [596] := 21.795, [597] := 22.13, [598] := 21.67, [599] := 21.65,
        [600] := 21.984999, [601] := 21.74, [602] := 21.885, [603] := 21.555, [604] := 22.029999, [605] := 21.92, [606] := 21.96, [607] := 21.619999, [608] := 22.085, [609] := 21.945, [610] := 21.9, [611] := 21.785, [612] := 21.664999, [613] := 22.145, [614] := 21.68, [615] := 21.83, [616] := 21.97, [617] := 22.02, [618] := 21.744999, [619] := 21.814999, [620] := 22.119999, [621] := 21.765, [622] := 22.21, [623] := 21.72, [624] := 22.119999, [625] := 21.945, [626] := 21.975, [627] := 21.76, [628] := 21.685, [629] := 22.164999, [630] := 21.725, [631] := 21.97, [632] := 21.74, [633] := 22.18, [634] := 22.17, [635] := 21.925, [636] := 21.945, [637] := 21.805, [638] := 22.24, [639] := 21.99, [640] := 21.955, [641] := 21.82, [642] := 22.255, [643] := 21.75, [644] := 21.82, [645] := 22.025, [646] := 22.064999, [647] := 22.175, [648] := 21.695, [649] := 22.14, [650] := 21.88, [651] := 22.005, [652] := 21.705, [653] := 22.119999, [654] := 21.994999, [655] := 21.77, [656] := 21.81, [657] := 21.65, [658] := 22.055, [659] := 21.585,
        [660] := 21.755, [661] := 21.84, [662] := 21.96, [663] := 22.08, [664] := 21.64, [665] := 22.029999, [666] := 21.89, [667] := 21.984999, [668] := 21.689999, [669] := 22.17, [670] := 22.125, [671] := 22.08, [672] := 21.805, [673] := 21.73, [674] := 22.189999, [675] := 21.975, [676] := 22.115, [677] := 21.715, [678] := 22.17, [679] := 22.025, [680] := 21.935, [681] := 21.855, [682] := 22.16, [683] := 22.164999, [684] := 21.765, [685] := 22.039999, [686] := 21.76, [687] := 22.15, [688] := 21.685, [689] := 21.835, [690] := 21.945, [691] := 22.029999, [692] := 22.125, [693] := 21.65, [694] := 22.105, [695] := 21.96, [696] := 21.859999, [697] := 21.645, [698] := 21.975, [699] := 21.975, [700] := 21.515, [701] := 21.66, [702] := 21.699999, [703] := 21.84, [704] := 21.55, [705] := 21.5, [706] := 21.965, [707] := 21.65, [708] := 21.805, [709] := 21.525, [710] := 21.939999, [711] := 21.925, [712] := 21.685, [713] := 21.785, [714] := 21.99, [715] := 22.085, [716] := 21.635, [717] := 21.89, [718] := 21.814999, [719] := 22.064999,
        [720] := 21.689999, [721] := 21.725, [722] := 22.015, [723] := 21.904999, [724] := 22.06, [725] := 21.715, [726] := 22.164999, [727] := 22.14, [728] := 21.904999, [729] := 21.895, [730] := 22.074999, [731] := 22.154999, [732] := 21.789999, [733] := 21.945, [734] := 21.76, [735] := 22.08, [736] := 21.645, [737] := 21.645, [738] := 22.01, [739] := 21.755, [740] := 21.914999, [741] := 21.64, [742] := 22.029999, [743] := 21.56, [744] := 21.59, [745] := 21.885, [746] := 21.705, [747] := 21.835, [748] := 21.484999, [749] := 21.9, [750] := 21.805, [751] := 21.619999, [752] := 21.664999, [753] := 21.59, [754] := 21.92, [755] := 21.814999, [756] := 22.035, [757] := 21.685, [758] := 22.185, [759] := 22.085, [760] := 21.984999, [761] := 21.8, [762] := 22.115, [763] := 22.145, [764] := 21.859999, [765] := 21.84, [766] := 21.71, [767] := 22.135, [768] := 21.779999, [769] := 21.96, [770] := 21.77, [771] := 22.16, [772] := 22.109999, [773] := 21.779999, [774] := 21.965, [775] := 22.085, [776] := 22.24, [777] := 21.865, [778] := 22.13, [779] := 21.935,
        [780] := 22.23, [781] := 21.744999, [782] := 22.185, [783] := 22.025, [784] := 21.865, [785] := 21.83, [786] := 21.675, [787] := 22.105, [788] := 21.74, [789] := 21.925, [790] := 21.725, [791] := 22.095, [792] := 21.765, [793] := 21.939999, [794] := 21.73, [795] := 22.109999, [796] := 22.08, [797] := 21.74, [798] := 21.939999, [799] := 21.619999, [800] := 22.074999, [801] := 21.615, [802] := 22.015, [803] := 21.55, [804] := 22.035, [805] := 21.605, [806] := 21.755, [807] := 21.755, [808] := 21.945, [809] := 22.07, [810] := 21.595, [811] := 22.039999, [812] := 21.789999, [813] := 21.925, [814] := 21.635, [815] := 21.615, [816] := 22.09, [817] := 21.715, [818] := 21.925, [819] := 21.855, [820] := 22.199999, [821] := 21.76, [822] := 21.9, [823] := 21.975, [824] := 22.05, [825] := 22.154999, [826] := 21.68, [827] := 22.095, [828] := 21.885, [829] := 21.93, [830] := 21.695, [831] := 21.595, [832] := 22.01, [833] := 21.705, [834] := 22.095, [835] := 21.64, [836] := 22.055, [837] := 21.795, [838] := 22.064999, [839] := 21.695,
        [840] := 22.14, [841] := 21.91, [842] := 21.97, [843] := 21.72, [844] := 21.625, [845] := 21.83, [846] := 21.965, [847] := 22.09, [848] := 21.64, [849] := 22.035, [850] := 21.779999, [851] := 21.925, [852] := 21.64, [853] := 22.0, [854] := 22.01, [855] := 21.615, [856] := 21.939999, [857] := 21.77, [858] := 21.975, [859] := 21.595, [860] := 21.755, [861] := 21.904999, [862] := 21.96, [863] := 22.145, [864] := 21.66, [865] := 22.085, [866] := 21.765, [867] := 22.05, [868] := 21.705, [869] := 22.164999, [870] := 21.955, [871] := 22.02, [872] := 21.785, [873] := 21.715, [874] := 22.195, [875] := 21.76, [876] := 22.085, [877] := 21.914999, [878] := 22.095, [879] := 21.765, [880] := 21.76, [881] := 22.109999, [882] := 21.939999, [883] := 22.095, [884] := 21.744999, [885] := 22.21, [886] := 22.09, [887] := 21.83, [888] := 21.76, [889] := 21.609999, [890] := 22.08, [891] := 21.785, [892] := 22.039999, [893] := 21.615, [894] := 22.085, [895] := 21.795, [896] := 21.975, [897] := 21.645, [898] := 22.074999, [899] := 22.045,
        [900] := 21.68, [901] := 21.93, [902] := 21.805, [903] := 22.09, [904] := 21.72, [905] := 21.75, [906] := 22.18, [907] := 21.904999, [908] := 22.08, [909] := 21.859999, [910] := 22.17, [911] := 21.715, [912] := 21.8, [913] := 21.859999, [914] := 22.039999, [915] := 22.1, [916] := 21.64, [917] := 21.949999, [918] := 21.779999, [919] := 21.98, [920] := 21.619999, [921] := 22.1, [922] := 21.99, [923] := 21.82, [924] := 21.84, [925] := 21.699999, [926] := 22.119999, [927] := 21.689999, [928] := 21.96, [929] := 21.775, [930] := 22.09, [931] := 22.13, [932] := 21.675, [933] := 22.035, [934] := 21.75, [935] := 22.035, [936] := 21.605, [937] := 21.58, [938] := 21.869999, [939] := 21.835, [940] := 21.695, [941] := 21.619999, [942] := 21.97, [943] := 21.779999, [944] := 21.939999, [945] := 21.6, [946] := 22.06, [947] := 21.97, [948] := 21.715, [949] := 21.814999, [950] := 21.68, [951] := 22.06, [952] := 21.619999, [953] := 21.715, [954] := 21.814999, [955] := 21.865, [956] := 21.574999, [957] := 21.58, [958] := 22.0, [959] := 21.81,
        [960] := 22.08, [961] := 21.64, [962] := 22.15, [963] := 21.865, [964] := 22.145, [965] := 21.755, [966] := 21.785, [967] := 22.045, [968] := 21.935, [969] := 21.845, [970] := 21.664999, [971] := 22.115, [972] := 21.664999, [973] := 21.77, [974] := 21.755, [975] := 21.914999, [976] := 22.015, [977] := 21.59, [978] := 21.945, [979] := 21.81, [980] := 21.975, [981] := 21.63, [982] := 21.654999, [983] := 22.01, [984] := 21.824999, [985] := 21.869999, [986] := 21.765, [987] := 22.189999, [988] := 22.119999, [989] := 21.875, [990] := 21.925, [991] := 22.055, [992] := 22.13, [993] := 21.765, [994] := 21.949999, [995] := 21.68, [996] := 22.09, [997] := 21.609999, [998] := 21.789999, [999] := 21.85);
   FE_4303_WEIGHT : REAL[100];
   FE_4304 : REAL := 1.725;
   FE_4304_AOI : Analog_Scale := (Analog_In := 4497.0, Offset_In := -4000.0, Analog_Min_In := 4000.0, Analog_Max_In := 20000.0, Analog_Max_Out := 50.0, Analog_Out := 1.553125);
   FE_4304_Low : REAL;
   FE_4304_OffSet : REAL := -4000.0;
   FE_4304_Sf : REAL := 0.002635564;
   FE_4305 : REAL := -1.779218;
   FE_4305_lOO : REAL;
   FE_4305_LOW : REAL;
   FE_4305_OffSet : REAL := 4000.0;
   FE_4305_Prop_Gain : DINT := 1;
   FE_4305_Sf : REAL := 0.010654;
   FilterChangePB : BOOL;
   FIT_4302_1 : AStd_AnalogInput := (Raw := 3948.0, Scaled := -0.4875, Scaling.RawMinS := 4000.0, Scaling.RawMaxS := 20000.0, Scaling.EngMaxS := 150.0, LowLow.LimitC := 5.0, LowLow.LimitOffSetC := 5.0, LowLow.Tmr.PRE := 15000, LowLow.Disabled := 1, Low.LimitC := 15.0, Low.Tmr.PRE := 15000, Low.Disabled := 1, High.LimitC := 80.0, High.Tmr.PRE := 15000, High.Disabled := 1, HighHigh.LimitC := 90.0, HighHigh.Tmr.PRE := 15000, HighHigh.Disabled := 1, Fault.LimitC := 3000.0, Fault.LimitOffSetC := 1000.0, Fault.Tmr.PRE := 10000, FaultReset := 500.0);
   FIT_4302_1_AOI : AStd_AI_AOI := (InputRaw_I := 3949.0, cfgRawMin := 4000.0, cfgRawMax := 20000.0, cfgEUMax := 150.0, Scaled := -0.47812498);
   FIT_4302_1_Holding : DINT := 3945;
   FIT_4302_1_sim_Val : DINT := 35;
   FIT_4302_1_Simulation : BOOL;
   FIT_4302_2 : AStd_AnalogInput := (Raw := 3939.0, Scaled := -0.7625, Scaling.RawMinS := 4000.0, Scaling.RawMaxS := 20000.0, Scaling.EngMaxS := 200.0, LowLow.LimitC := 10.0, LowLow.LimitOffSetC := 10.0, LowLow.Tmr.PRE := 30000, LowLow.Disabled := 1, Low.LimitC := 15.0, Low.Tmr.PRE := 30000, Low.Disabled := 1, High.LimitC := 80.0, High.Tmr.PRE := 30000, High.Disabled := 1, HighHigh.LimitC := 90.0, HighHigh.Tmr.PRE := 30000, HighHigh.Disabled := 1, Fault.LimitC := 3000.0, Fault.LimitOffSetC := 1000.0, Fault.Tmr.PRE := 5000, FaultReset := 500.0);
   FIT_4302_2_AOI : AStd_AI_AOI := (InputRaw_I := 3939.0, cfgRawMin := 4000.0, cfgRawMax := 20000.0, cfgEUMax := 200.0, Scaled := -0.7625, CommsStatus := 1);
   FIT_4302_2_Holding : DINT := 3939;
   FIT_4302_2_Samples : DINT := 100;
   FIT_4302_2_sim_Val : DINT := 40;
   FIT_4302_2_Simulation : BOOL := 1;
   FIT_4305_xx : AStd_AnalogInput := (Raw := 3948.0, Scaled := -1.3000001, Scaling.RawMinS := 4000.0, Scaling.RawMaxS := 20000.0, Scaling.EngMaxS := 400.0, LowLow.LimitC := 10.0, LowLow.LimitOffSetC := 1.0, LowLow.Tmr.PRE := 60000, LowLow.Disabled := 1, Low.LimitC := 30.0, Low.Tmr.PRE := 30000, Low.Disabled := 1, High.LimitC := 170.0, High.Tmr.PRE := 30000, High.Disabled := 1, HighHigh.LimitC := 180.0, HighHigh.Tmr.PRE := 30000, HighHigh.Disabled := 1, Fault.LimitC := 3000.0, Fault.LimitOffSetC := 1000.0, Fault.Tmr.PRE := 5000, FaultReset := 500.0);
   FIT_4305_xx_AOI : AStd_AI_AOI := (InputRaw_I := 3951.0, cfgRawMin := 4000.0, cfgRawMax := 20000.0, cfgEUMax := 400.0, Scaled := -1.225, CommsStatus := 1);
   FIT_4305_xx_Holding : DINT := 3945;
   FIT_4305_xx_Samples : DINT := 100;
   FIT_4305_xx_sim_Val : DINT := 50;
   FIT_4305_xx_Simulation : BOOL := 1;
   FIT_S47_1 : AStd_AnalogInput := (Raw := 4261.0, Scaled := 8.15625, Scaling.RawMinS := 4000.0, Scaling.RawMaxS := 20000.0, Scaling.EngMaxS := 500.0, LowLow.Tmr.PRE := 1000, Low.Tmr.PRE := 1000, High.LatchA := 1, High.DetectS := 1, High.BitS := 1, High.Tmr.PRE := 1000, High.Tmr.ACC := 1013, High.Tmr.EN := 1, High.Tmr.DN := 1, HighHigh.LatchA := 1, HighHigh.DetectS := 1, HighHigh.BitS := 1, HighHigh.Tmr.PRE := 1000, HighHigh.Tmr.ACC := 1013, HighHigh.Tmr.EN := 1, HighHigh.Tmr.DN := 1, Fault.LimitC := 4000.0, Fault.Tmr.PRE := 1000);
   FIT_S47_1_AOI : AStd_AI_AOI := (InputRaw_I := 4258.0, cfgRawMin := 4000.0, cfgRawMax := 20000.0, cfgEUMax := 500.0, Scaled := 8.0625);
   FIT_S47_1MassFlowLBMin : REAL := 8.3125;
   FIT_S47_1PulseCounter : COUNTER := (PRE := 50000);
   FLH : REAL := 18.0;
   FLL : REAL := 6.0;
   FlowmeterPulse : BOOL := 1;
   Found : DINT;
   FQIC_4302_11_AOI : Analog_Scale := (Offset_In := -4000.0, Analog_Min_In := 4000.0, Analog_Max_In := 20000.0, Analog_Max_Out := 80.0, Analog_Out := -20.0);
   FQIC_4302_11_Calc_TransferSetpoint : DINT := 44000;
   FQIC_4302_11_Corrected : REAL := -20.0;
   FQIC_4302_11_Correction_Sf : REAL := 1.0;
   FQIC_4302_11_Correction_Sf_DELETEME : DINT;
   FQIC_4302_11_CurrentAmount : DINT;
   FQIC_4302_11_CurrentTrasferredLb : DINT := 2385;
   FQIC_4302_11_Flow_Raw : DINT;
   FQIC_4302_11_OffSet_Out : REAL;
   FQIC_4302_11_Out : REAL := -20.0;
   FQIC_4302_11_Pulse : BOOL;
   FQIC_4302_11_PulseCounter : COUNTER := (PRE := 890000000, ACC := 477);
   FQIC_4302_11_PulseToLbFactor : DINT := 5;
   FQIC_4302_11_Reset : BOOL;
   FQIC_4302_11_TargetAmount : DINT;
   FQIC_4302_11_TransferOffset : DINT := 100;
   FQIC_4302_11_TransferSetpoint : DINT := 44000;
   FQIC_4302_11_TransferStopValueLb : DINT := 43900;
   From_Main : MESSAGE;
        MessageParameters(ServiceCode := 16#004c, LocalElement := Main_to_Dispersion, ...)
   From_Main2 : MESSAGE;
        MessageParameters(ServiceCode := 16#004c, LocalElement := Main_to_Dispersion2, ...)
   From_Sil2 : MESSAGE;
        MessageParameters(ServiceCode := 16#004c, LocalElement := SIL2_to_Dispersion, ...)
   From_Sil2_Analog : MESSAGE;
        MessageParameters(ServiceCode := 16#004c, LocalElement := SIL2_to_Dispersion_Analog[0], ...)
   FromControlRoomPLC : MESSAGE;
   FV_4305_xx : AStd_VlvModulating := (AutoC := 1, AutoS := 1, AutoCtrlS := 1, Perm.IntlkS := 1, Perm.SafeS := 1, ManPosC := 50.0, AutoCtrlC := 4, AutoPosC[1] := 100.0, AutoPosC[2] := 50.0, AutoPosS := 50.0, ScaledO := 50.0, Scaling.RawMinS := 4000.0, Scaling.RawMaxS := 20000.0, Scaling.EngMaxS := 100.0, RawO := 12000.0);
   FV_4305_xx_AOI : AStd_VlVModulating_AOI := (cfgEUMax := 100.0, cfgRawMin := 4000.0, cfgRawMax := 20000.0, OutputRaw_O := 12000.0, AutoS := 1, OpenS := 1);
   GasAlarmTmr : TIMER := (PRE := 40000);
   GasAlarmTmrOff : TIMER := (PRE := 1000);
   GasAlarmTmrOn : TIMER := (PRE := 2000);
   GenPurp : AStd_GeneralPurp := (AlwaysOn := 1, PowerUpDelay := 1, AlternateScan := 1, HalfSecondSquare := 1, OneSecondSquare := 1, Tmr[0].PRE := 500, Tmr[0].ACC := 515, Tmr[0].EN := 1, Tmr[0].DN := 1, Tmr[1].PRE := 500, Tmr[1].ACC := 435, Tmr[1].EN := 1, Tmr[1].TT := 1, Tmr[2].PRE := 1000, Tmr[2].ACC := 342, Tmr[2].EN := 1, Tmr[2].TT := 1, ONS := 1);
   GLOBAL_RESET : BOOL;
   Heat_Setpoint_4301 : DINT := 150;
   Heat_Setpoint_4302 : DINT := 150;
   Heat_SP : REAL := 22.0;
   hfdhh : BOOL;
   hhh : BOOL := 1;
   HHI_Process_Temp_Alarm_4302 : BOOL;
   HMI_4303_Timer : REAL := 5.0;
   HMI_4304_Timer : REAL := 60.0;
   HMI_Cat_Isolation_T430X_Timer : REAL;
   HMI_Cat_Isolation_Valve_Timer : REAL := 2.0;
   HMI_Drum_Addition_T430X_Timer : REAL := 30.0;
   HMI_Drum_Addition_Timer : REAL := 120.0;
   HMI_Linked_Timer : REAL := 30.0;
   HMI_Mon_Isolation_K400_Timer : REAL := 3.0;
   HMI_Mon_Isolation_T430X_Timer : REAL;
   HMI_V4304_PumpSpeedScaleIn : REAL := 152.0;
   Hold_For_Flow_Switch : BOOL;
   Hold_For_Pump_Enable : BOOL;
   HornONS_Phases : BOOL[32];
   HS_9A249 : ALIAS FOR Local:1:O.Data[0].17;
   HS_9A640 : ALIAS FOR Local:1:O.Data[0].18;
   HS_S51_1 : AStd_DiscreteInput := (InI := 1, Alm.LatchA := 1, Alm.DetectS := 1, Alm.BitS := 1, Alm.Tmr.ACC := 17, Alm.Tmr.EN := 1, Alm.Tmr.DN := 1);
   HS_S51_1_AOI : AStd_DI_AOI := (Input_I := 1, cfgDebounceTmrPre := 1000, cfgAlarmEnable := 1, AlmS := 1);
   HS_S51_1_IRaw : BOOL := 1;
   HS_S51_1_Simulation : BOOL := 1;
   HS_S51_2 : AStd_DiscreteInput := (InI := 1, Alm.LatchA := 1, Alm.DetectS := 1, Alm.BitS := 1, Alm.Tmr.ACC := 14, Alm.Tmr.EN := 1, Alm.Tmr.DN := 1);
   HS_S51_2_AOI : AStd_DI_AOI := (Input_I := 1, cfgDebounceTmrPre := 1000, cfgAlarmEnable := 1, AlmS := 1);
   HS_S51_2_IRaw : BOOL;
   HS_S51_2_Simulation : BOOL := 1;
   InRawScaledMelimine : INT;
   INTERLOCK_TEST_BUTTON_1 : BOOL;
   INTERLOCK_TEST_BUTTON_2 : BOOL;
   INTERLOCK_TEST_BUTTON_3 : BOOL;
   INTERLOCK_TEST_BUTTON_3_ONS : BOOL;
   INX_Alarm : BOOL[32];
   Inx_AlarmScanIdx : DINT := 11;
   INX_AlarmTmr : TIMER[32] := ([0].PRE := 15000, [1].PRE := 15000, [2].PRE := 15000, [3].PRE := 15000, [4].PRE := 15000);
   Inx_Alr_To_Sound_Horn : BOOL[128] := ([2] := 1, [7] := 1, [17] := 1, [18] := 1, [21] := 1, [22] := 1);
   INX_ALRM_BUZ : ALIAS FOR Local:1:O.Data[1].9;
   InxAlarmResetBit : BOOL;
   InxAlarms : BOOL[128] := ([11] := 1);
   jde_test : BOOL;
   JHAKJHKL : BOOL;
   K200_PhaseTransfer : AStd_PLI := (IdleS := 1, CurrentStateCodeS := 1, PreventStartS := 4, AlarmS := 4, StepNo := 1, StepBit := 2, RealParameters[0] := 1063.6019, RealParameters[1] := 20807.328, DINTParameters[0] := 2, PreventStartInhibitC := 127, AlarmInhibitC := 63, IntSafDisp := 4, InterlockTimers.Timers[3].PRE := 3000);
   K200_PhaseTransfer_AOI : AStd_PLI_AOI := (PreventStartS := 1, AlmS := 1, StepNo := 1, cfgAutoReset := 1);
   K200_PhaseTransfer_StepComplete : BOOL[32];
   K2_Temperature_Alarm_Enable_Bit : BOOL;
   K400_PhaseTransfer : AStd_PLI := (IdleS := 1, CurrentStateCodeS := 1, PreventStartS := 132, AlarmS := 4, StepNo := 1, StepBit := 2, RealParameters[0] := 38078.19, RealParameters[1] := -15557.379, DINTParameters[0] := 3, DINTParameters[1] := 1800, DINTParameters[19] := 3, PreventStartInhibitC := 511, AlarmInhibitC := 383, IntSafDisp := 132, InterlockTimers.Timers[3].PRE := 3000);
   K400_PhaseTransfer_AOI : AStd_PLI_AOI := (PreventStartS := 1, AlmS := 1, StepNo := 1, cfgAutoReset := 1);
   K400_PhaseTransfer_StepComplete : BOOL[32];
   K4_High_Temp : BOOL;
   K4_Low_Temp : BOOL;
   LAH_4302_11 : BOOL;   // Truck Loading Level Alarm High Probe
   LAH_S4352_1 : ALIAS FOR Local:1:I.Data[27].13;
   LastScannedCode : STRING := '75381';
   LastTrasferredLb : REAL;
   LevelAlarmBeaconsRelay : BOOL;
   limitswitch : BOOL := 1;
   Linked_Timer : TIMER := (PRE := 30000);
   LS_200_1_IRaw : REAL := 50.0;
   LS_200_1_sim_Val : DINT := 50;
   LS_200_1_Simulation : BOOL := 1;
   LS_26_H : TIMER := (PRE := 10000);
   LS_26_H_Alarm : BOOL;
   LS_26_High : BOOL;
   LS_28_H : TIMER := (PRE := 10000);
   LS_28_H_Alarm : BOOL;
   LS_400_1_IRaw : REAL := 50.0;
   LS_400_1_sim_Val : DINT := 50;
   LS_400_1_Simulation : BOOL := 1;
   LS_4301 : ALIAS FOR Local:2:I.Data.10;
   LS_4301_High : BOOL;
   LS_4302 : ALIAS FOR Local:2:I.Data.11;
   LS_4302_1_H : TIMER := (PRE := 2000);
   LS_4302_Dry : DINT := 9;
   LS_4302_Faulted : BOOL;
   LS_4302_H_Off_Timer : TIMER := (PRE := 10000);
   LS_4302_H_Timer : TIMER := (PRE := 10000);
   LS_4302_High : BOOL;
   LS_4302_Raw : INT := 8064;
   LS_4302_Wet : REAL := 15.0;
   LS_4320 : ALIAS FOR Local:1:I.Data[4].4;
   LS_S51_1 : AStd_DiscreteInput := (Alm.Tmr.PRE := 2000);
   LS_S51_1_AOI : AStd_DI_AOI := (cfgDebounceTmrPre := 1000, cfgAlarmEnable := 1);
   LS_S51_1_IRaw : BOOL;
   LS_S51_1_Simulation : BOOL;
   LS_T51_High : ALIAS FOR Local:1:I.Data[27].14;
   LS_T53_High : ALIAS FOR Local:1:I.Data[27].12;
   LVL_W2_High : ALIAS FOR Local:1:I.Data[1].22;
   LVL_W4_High : ALIAS FOR Local:1:I.Data[1].23;
   Main_from_Dispersion : DINT;
   Main_from_Dispersion2 : DINT;
   Main_to_Dispersion : DINT;
   Main_to_Dispersion2 : DINT;
   MAINT_SV4303_03_PB : BOOL;
   MAINT_SV4303_04_PB : BOOL;
   MAINT_SV4304_02_PB : BOOL;
   MAINT_SV4304_03_PB : BOOL;
   MAINT_XV4303_05_PB : BOOL;
   MAINT_XV4304_04_PB : BOOL;
   MaxHeatTmr4301 : TIMER;
   MaxHeatTmr4302 : TIMER := (PRE := 900000);
   MCC1D4_20_TT5_Relay : BOOL := 1;
   MCC1F3_TT1_Relay : BOOL := 1;
   MCC1F4_8_TT9_Relay : BOOL := 1;
   MCR_Bulk : ALIAS FOR Local:1:I.Data[33].4;
   Melamine_Amount_Per_Count : REAL := 5.0;
   Melamine_Charge_Remaining : REAL := -1.0;
   Melamine_Flow_Rate : REAL;
   Melamine_Flow_Raw : INT := -29848;
   Melamine_Flow_Raw_Adjusted : REAL := 19.0;
   Melamine_Flow_Scale_Factor : REAL := 0.008496176;
   Melamine_Last_Charge : REAL := 10715.0;
   Melamine_MA : REAL;
   Melamine_Manual_Start : BOOL;
   Melamine_Pump_Off : BOOL;
   Melamine_Pump_Run : BOOL;
   Melamine_Transfer : BOOL;
   Melamine_transfer_amount : REAL;
   melamine_transfer_setpoint : REAL := 10714.0;
   MelaminePumpTmr : TIMER := (PRE := 500);
   Melimine_Max_Flow : DINT := 500;
   Melimine_Pump_Manual_Run : BOOL;
   Messaging_Timer : TIMER := (PRE := 4000, ACC := 541, EN := 1, TT := 1);
   Micro_Motion : COUNTER := (PRE := 2000000, ACC := 1, CU := 1);
   micromotio_tmr : TIMER;
   micromotion : TIMER := (PRE := 100);
   MICROMOTION_COUNT : DINT;
   MICROMOTION_POUNDS : REAL := 5.0;
   MICROMOTION_PULSE_COUNT_COUNT_INPUT : ALIAS FOR Local:1:I.Data[32].1;
   MICROMOTION_SF : REAL := 5.0;
   MIRCOMOITION_ENABLE : ALIAS FOR Local:1:I.Data[32].7;
   MIXER_A_4301_RUN : ALIAS FOR Local:1:O.Data[0].0;
   MIXER_A_4303_AUX : ALIAS FOR Local:1:I.Data[1].4;
   MIXER_A_4303_RUN : ALIAS FOR Local:1:O.Data[0].4;
   MIXER_A_4304_AUX : ALIAS FOR Local:1:I.Data[1].16;
   MIXER_A_4304_RUN : ALIAS FOR Local:1:O.Data[0].16;
   MIXER_A_4320_AUX : ALIAS FOR Local:1:I.Data[1].5;
   MIXER_A_4320_RUN : ALIAS FOR Local:1:O.Data[0].5;
   MIXER_T_4301_AUX : ALIAS FOR Local:1:I.Data[1].0;
   MM_Gal_Ach : ALIAS FOR Local:1:I.Data[32].2;
   MMI_7_8_Transfer_Pump_Start : BOOL;
   MMI_7_8_Transfer_Pump_Stop : BOOL;
   MMI_A_4301_01_RUN_PB : BOOL;
   MMI_A_4301_02_RUN_PB : BOOL;
   MMI_A_4302_RUN_PB : BOOL;
   MMI_A_4303_RUN_PB : BOOL;
   MMI_A_4304_RUN_PB : BOOL;
   MMI_A_4320_RUN_PB : BOOL;
   MMI_AIR_PURGE_4301_PB : BOOL;
   MMI_AIR_PURGE_4302_PB : BOOL;
   MMI_B4320_Level : INT := 67;
   MMI_Cat_Man_Req : BOOL;
   MMI_Cat_Nit_Purge_Time : REAL := 7.0;
   MMI_Cat_Recirc_Pump_Speed : REAL := 100.0;
   MMI_COOL_DISH_4301_PB : BOOL;
   MMI_COOL_DISH_4302_PB : BOOL;
   MMI_COOL_VALVE_4301_PB : BOOL;
   MMI_COOL_VALVE_4302_PB : BOOL;
   MMI_Disp_Alarm_Reset_Pb : BOOL;
   MMI_Dispersion_Interlock_Bypass : BOOL;
   MMI_Dispersion_Interlock_Bypass_pb : BOOL;
   MMI_INX_Alarm_Reset_Pb : BOOL;
   MMI_INX_Solvent_Bypass : BOOL;
   MMI_INX_Solvent_Bypass_TOG : BOOL := 1;
   MMI_K2_TransTime_SP : REAL;
   MMI_K2_Weight_SP : REAL;
   MMI_Mixer_T52_RUN_PB : BOOL;
   MMI_Mixer_T53_RUN_PB : BOOL;
   MMI_Mon_Man_Req : BOOL;
   MMI_Mon_Nit_Purge_Time : REAL := 10.0;
   MMI_Mon_Recirc_Pump_Speed : REAL := 100.0;
   MMI_P_4301_RUN_PB : BOOL;
   MMI_P_4302_RUN_PB : BOOL;
   MMI_P_4303_Run_Pb : BOOL;
   MMI_P_4304_RUN_PB : BOOL;
   MMI_P_4305_RUN_PB : BOOL;
   MMI_P_4320_RUN_PB : BOOL;
   MMI_RO_Acc_Weight_Reset : BOOL;
   MMI_RO_TransTime_SP : REAL := 2.0;
   MMI_RO_Weight_SP : REAL := 200.0;
   MMI_SOL_SV_4303_01 : BOOL;
   MMI_SOL_SV_4303_02 : BOOL;
   MMI_SOL_SV_4303_03 : BOOL;
   MMI_SOL_SV_4304 : BOOL;
   MMI_SOL_XV_4301 : BOOL;
   MMI_SOL_XV_4302 : BOOL;
   MMI_SOL_XV_4303 : BOOL;
   MMI_SOL_XV_4304 : BOOL;
   MMI_SOL_XV_4320 : BOOL;
   MMI_SV4303_03_PB : BOOL;
   MMI_SV4303_04_PB : BOOL;
   MMI_SV4304_02_PB : BOOL;
   MMI_SV4304_03_PB : BOOL;
   MMI_SV4304_PB : BOOL;
   MMI_T4301_AIR_PURGE_REQUEST : BOOL;
   MMI_T4301_Level : INT;
   MMI_T4302_AIR_PURGE_REQUEST : BOOL;
   MMI_T4302_Level : INT;
   MMI_T51_Level : INT := 65;
   MMI_T52_Level : INT := 93;
   MMI_T52_WARN_BYPASS : BOOL;
   MMI_T53_Level : INT := 55;
   MMI_T53_WARN_BYPASS : BOOL;
   MMI_THINNING_LOADING_VALVE : BOOL;
   MMI_V4301_Mixer_SP : REAL;
   MMI_V4302_Mixer_SP : REAL;
   MMI_V4303_Acc_Weight_Reset : BOOL;
   MMI_V4303_TransTime_SP : REAL := 360.0;
   MMI_V4303_Weight_SP : REAL := 7800.0;
   MMI_V4304_Acc_Weight : REAL := 67.053314;
   MMI_V4304_Acc_Weight_Temp : REAL := 67.053314;
   MMI_V4304_TransTime_SP : REAL := 400.0;
   MMI_V4304_Weight_SP : REAL := 630.0;
   MMI_W4303_Acc_Weight : REAL := 859.7244;
   MMI_W4303_Level : INT := 48;
   MMI_XV4303_03_PB : BOOL;
   MMI_XV4303_04_PB : BOOL;
   MMI_XV4303_05_PB : BOOL;
   MMI_XV4304_02_PB : BOOL;
   MMI_XV4304_03_PB : BOOL;
   MMI_XV4304_04_PB : BOOL;
   MMI_XV4304_PB : BOOL;
   MMI_XV_4301_PB : BOOL;
   MMI_XV_4302_PB : BOOL;
   MMI_XV_4304_01_PB : BOOL;
   MMI_XV_4320_1_PB : BOOL;
   MMI_XV_4320_2_PB : BOOL;
   MMI_XV_5201_PB : BOOL;
   MMI_XV_5202_PB : BOOL;
   MMI_XV_5301_PB : BOOL;
   MMI_XV_5302_PB : BOOL;
   MMI_Z1H_4301_PB : BOOL;
   MMI_Z1H_4302_PB : BOOL;
   MMI_Z2H_4301_PB : BOOL;
   MMI_Z2H_4302_PB : BOOL;
   MMI_ZH3_4301_PB : BOOL;
   MMI_ZH3_4302_PB : BOOL;
   Momomer_Ons : DINT;
   Mon_Bogus_Bit : BOOL;
   Mon_Destination_K400 : BOOL := 1;
   Mon_Destination_K400_ONS : BOOL;
   Mon_Destination_K400_PB : BOOL;
   Mon_Destination_T4301 : BOOL;
   Mon_Destination_T4301_ONS : BOOL;
   Mon_Destination_T4301_PB : BOOL;
   Mon_Destination_T4302 : BOOL;
   Mon_Destination_T4302_ONS : BOOL;
   Mon_Destination_T4302_PB : BOOL;
   Mon_Isolation_K400_Timer : TIMER := (PRE := 180000);
   Mon_Isolation_T430X_Timer : TIMER;
   Mon_Man_ONS : BOOL;
   Mon_Pump_Manual : BOOL;
   Mon_Purge_T430X_End_Timer : TIMER := (PRE := 5000);
   Mon_Purge_Transfer_K400 : Seq64 := (Sq.Step[0] := 1);
   Mon_Purge_Transfer_K400_ONS : BOOL;
   Mon_Purge_Transfer_T430X : Seq64 := (Sq.Step[0] := 1);
   Mon_Recirc_Transfer_K400 : Seq64 := (Val := 6, Sq.Step[6] := 1);
   Mon_Recirc_Transfer_T430X : Seq64 := (Sq.Step[1] := 1);
   Mon_Scale_Factor : REAL := 0.0031135;
   Mon_Tank_Destination : DINT := 1;
   MON_VALV_ENBL : DINT := 1;
   MON_VALV_ENBL_BIT1 : BOOL := 1;
   MON_VALV_ENBL_PB1 : BOOL;
   Mon_Zero : REAL := 4000.0;
   Monomer_Barcode : STRING;
   Monomer_Barcode_Last : STRING;
   Monomer_Barcode_Scan_Index : DINT;
   Monomer_Barcode_Search : BOOL;
   Monomer_Destination : DINT;
   Monomer_Fill_Pump_Running : BOOL;
   Monomer_Fill_Pump_Stopped : BOOL;
   Monomer_Flow_Start_Timer : TIMER := (PRE := 5000);
   Monomer_Flow_Stop_Timer : TIMER := (PRE := 5000);
   Monomer_MaxFeedRate : REAL := 46.0;
   MONOMER_RESET : BOOL;
   Monomer_Scanner_Reset_Timer : TIMER := (PRE := 5000);
   MonomerTimers_0_HMI : REAL := 10.006;
   New_DispertionAlarmDetected : BOOL;
   NEW_TO : MESSAGE;
        MessageParameters(ServiceCode := 16#004c, LocalElement := TO_ALARM_MSG_DINT, ...)
   NM_4303_AOI : AStd_AI_AOI := (InputRaw_I := 17151.4, cfgRawMin := 4000.0, cfgRawMax := 20000.0, cfgEUMax := 25.0, Scaled := 20.549063);
   NM_4303_O2 : AStd_AnalogInput := (Raw := 17157.5, Scaled := 20.558594, Scaling.RawMinS := 4000.0, Scaling.RawMaxS := 20000.0, Scaling.EngMaxS := 25.0, LowLow.LimitC := 3.0, LowLow.Tmr.PRE := 1000, High.LatchA := 1, High.DetectS := 1, High.BitS := 1, High.Tmr.PRE := 1000, High.Tmr.ACC := 1006, High.Tmr.EN := 1, High.Tmr.DN := 1, HighHigh.LimitC := 22.0, HighHigh.Tmr.PRE := 1000, Fault.LimitC := 4000.0);
   NM_4303_O2_SIGNAL : REAL := 17155.32;
   NM_4303_SIGNAL_AVERAGE : MOVING_AVERAGE := (In := 17150.0, SampleEnable := 1, NumberOfSamples := 50, Out := 17158.2);
   NM_4303_SIGNAL_AVERAGE_STORAGE : REAL[1000] := ([0] := 17293.0, [1] := 17052.0, [2] := 17214.0, [3] := 17047.0, [4] := 17298.0, [5] := 17208.0, [6] := 17158.0, [7] := 17094.0, [8] := 17012.0, [9] := 17307.0, [10] := 17011.0, [11] := 17264.0, [12] := 17168.0, [13] := 17193.0, [14] := 17058.0, [15] := 16999.0, [16] := 17300.0, [17] := 17029.0, [18] := 17122.0, [19] := 17128.0, [20] := 17278.0, [21] := 17302.0, [22] := 17024.0, [23] := 17244.0, [24] := 17137.0, [25] := 17223.0, [26] := 17038.0, [27] := 17021.0, [28] := 17247.0, [29] := 17107.0, [30] := 17147.0, [31] := 17044.0, [32] := 17295.0, [33] := 16998.0, [34] := 17037.0, [35] := 17217.0, [36] := 17138.0, [37] := 17242.0, [38] := 16998.0, [39] := 17297.0, [40] := 17224.0, [41] := 17188.0, [42] := 17054.0, [43] := 16996.0, [44] := 17297.0, [45] := 17074.0, [46] := 17168.0, [47] := 17056.0, [48] := 17281.0, [49] := 16998.0, [50] := 17026.0, [51] := 17235.0, [52] := 17114.0, [53] := 17228.0, [54] := 17031.0, [55] := 17298.0, [56] := 17289.0, [57] := 17047.0, [58] := 17208.0, [59] := 17043.0,
        [60] := 17293.0, [61] := 16998.0, [62] := 17089.0, [63] := 17156.0, [64] := 17203.0, [65] := 17048.0, [66] := 17104.0, [67] := 17140.0, [68] := 17219.0, [69] := 17297.0, [70] := 17018.0, [71] := 17246.0, [72] := 17141.0, [73] := 17269.0, [74] := 17004.0, [75] := 17015.0, [76] := 17255.0, [77] := 17156.0, [78] := 17090.0, [79] := 17007.0, [80] := 17305.0, [81] := 17049.0, [82] := 17152.0, [83] := 17096.0, [84] := 17257.0, [85] := 17308.0, [86] := 17009.0, [87] := 17273.0, [88] := 17052.0, [89] := 17293.0, [90] := 17000.0, [91] := 17299.0, [92] := 17228.0, [93] := 17134.0, [94] := 17120.0, [95] := 17001.0, [96] := 17302.0, [97] := 17032.0, [98] := 17119.0, [99] := 17129.0, [100] := 17234.0, [101] := 17303.0, [102] := 17074.0, [103] := 17183.0, [104] := 17074.0, [105] := 17276.0, [106] := 17006.0, [107] := 17021.0, [108] := 17251.0, [109] := 17101.0, [110] := 17149.0, [111] := 17043.0, [112] := 17296.0, [113] := 17000.0, [114] := 17040.0, [115] := 17223.0, [116] := 17135.0, [117] := 17291.0, [118] := 17001.0, [119] := 17301.0,
        [120] := 17105.0, [121] := 17255.0, [122] := 17016.0, [123] := 17307.0, [124] := 17224.0, [125] := 17135.0, [126] := 17116.0, [127] := 17026.0, [128] := 17305.0, [129] := 17003.0, [130] := 17188.0, [131] := 17066.0, [132] := 17284.0, [133] := 17304.0, [134] := 17068.0, [135] := 17183.0, [136] := 17074.0, [137] := 17274.0, [138] := 17005.0, [139] := 17304.0, [140] := 17253.0, [141] := 17098.0, [142] := 17085.0, [143] := 17010.0, [144] := 17308.0, [145] := 17108.0, [146] := 17222.0, [147] := 17039.0, [148] := 17298.0, [149] := 17256.0, [150] := 17102.0, [151] := 17154.0, [152] := 17013.0, [153] := 17310.0, [154] := 17016.0, [155] := 17267.0, [156] := 17102.0, [157] := 17260.0, [158] := 17014.0, [159] := 17041.0, [160] := 17220.0, [161] := 17142.0, [162] := 17292.0, [163] := 17001.0, [164] := 17299.0, [165] := 17226.0, [166] := 17261.0, [167] := 17013.0, [168] := 17309.0, [169] := 17267.0, [170] := 17152.0, [171] := 17104.0, [172] := 17020.0, [173] := 17312.0, [174] := 17012.0, [175] := 17086.0, [176] := 17180.0, [177] := 17190.0, [178] := 17288.0, [179] := 17009.0,
        [180] := 17312.0, [181] := 17130.0, [182] := 17246.0, [183] := 17035.0, [184] := 17311.0, [185] := 17247.0, [186] := 17126.0, [187] := 17142.0, [188] := 17010.0, [189] := 17310.0, [190] := 17029.0, [191] := 17241.0, [192] := 17032.0, [193] := 17310.0, [194] := 17291.0, [195] := 17120.0, [196] := 17141.0, [197] := 17043.0, [198] := 17304.0, [199] := 17026.0, [200] := 17255.0, [201] := 17154.0, [202] := 17216.0, [203] := 17050.0, [204] := 17005.0, [205] := 17303.0, [206] := 17096.0, [207] := 17209.0, [208] := 17059.0, [209] := 17295.0, [210] := 17216.0, [211] := 17154.0, [212] := 17109.0, [213] := 17021.0, [214] := 17312.0, [215] := 17012.0, [216] := 17278.0, [217] := 17117.0, [218] := 17249.0, [219] := 17024.0, [220] := 17155.0, [221] := 17101.0, [222] := 17261.0, [223] := 17201.0, [224] := 17166.0, [225] := 17088.0, [226] := 17004.0, [227] := 17191.0, [228] := 17180.0, [229] := 17078.0, [230] := 17011.0, [231] := 17290.0, [232] := 17068.0, [233] := 17173.0, [234] := 17091.0, [235] := 17308.0, [236] := 17293.0, [237] := 17061.0, [238] := 17146.0, [239] := 17042.0,
        [240] := 17304.0, [241] := 17005.0, [242] := 17303.0, [243] := 17226.0, [244] := 17141.0, [245] := 17123.0, [246] := 17028.0, [247] := 17311.0, [248] := 17009.0, [249] := 17195.0, [250] := 17072.0, [251] := 17286.0, [252] := 17312.0, [253] := 17026.0, [254] := 17257.0, [255] := 17160.0, [256] := 17271.0, [257] := 17015.0, [258] := 17313.0, [259] := 17273.0, [260] := 17092.0, [261] := 17171.0, [262] := 17065.0, [263] := 17290.0, [264] := 17006.0, [265] := 17029.0, [266] := 17189.0, [267] := 17291.0, [268] := 17304.0, [269] := 17034.0, [270] := 17180.0, [271] := 17068.0, [272] := 17284.0, [273] := 17006.0, [274] := 17309.0, [275] := 17251.0, [276] := 17111.0, [277] := 17147.0, [278] := 17005.0, [279] := 17287.0, [280] := 17062.0, [281] := 17232.0, [282] := 17035.0, [283] := 17305.0, [284] := 17248.0, [285] := 17116.0, [286] := 17139.0, [287] := 17228.0, [288] := 17284.0, [289] := 17069.0, [290] := 17194.0, [291] := 17036.0, [292] := 17308.0, [293] := 17027.0, [294] := 17116.0, [295] := 17026.0, [296] := 17309.0, [297] := 17284.0, [298] := 17066.0, [299] := 17199.0,
        [300] := 17087.0, [301] := 17271.0, [302] := 17013.0, [303] := 17310.0, [304] := 17262.0, [305] := 17094.0, [306] := 17168.0, [307] := 17057.0, [308] := 17289.0, [309] := 17002.0, [310] := 17140.0, [311] := 17110.0, [312] := 17249.0, [313] := 17307.0, [314] := 17006.0, [315] := 17284.0, [316] := 17198.0, [317] := 17171.0, [318] := 17085.0, [319] := 17275.0, [320] := 17310.0, [321] := 17018.0, [322] := 17259.0, [323] := 17166.0, [324] := 17263.0, [325] := 17016.0, [326] := 17013.0, [327] := 17221.0, [328] := 17145.0, [329] := 17252.0, [330] := 17023.0, [331] := 17303.0, [332] := 17233.0, [333] := 17128.0, [334] := 17132.0, [335] := 17233.0, [336] := 17306.0, [337] := 17004.0, [338] := 17292.0, [339] := 17142.0, [340] := 17225.0, [341] := 17043.0, [342] := 17128.0, [343] := 17130.0, [344] := 17234.0, [345] := 17308.0, [346] := 17025.0, [347] := 17250.0, [348] := 17149.0, [349] := 17218.0, [350] := 17046.0, [351] := 17299.0, [352] := 17207.0, [353] := 17163.0, [354] := 17093.0, [355] := 17016.0, [356] := 17297.0, [357] := 17048.0, [358] := 17145.0, [359] := 17113.0,
        [360] := 17248.0, [361] := 17307.0, [362] := 17004.0, [363] := 17282.0, [364] := 17190.0, [365] := 17170.0, [366] := 17085.0, [367] := 17303.0, [368] := 17287.0, [369] := 17056.0, [370] := 17207.0, [371] := 17040.0, [372] := 17299.0, [373] := 17000.0, [374] := 17101.0, [375] := 17150.0, [376] := 17214.0, [377] := 17294.0, [378] := 17000.0, [379] := 17297.0, [380] := 17226.0, [381] := 17199.0, [382] := 17056.0, [383] := 17290.0, [384] := 17304.0, [385] := 17079.0, [386] := 17177.0, [387] := 17073.0, [388] := 17308.0, [389] := 17007.0, [390] := 17072.0, [391] := 17192.0, [392] := 17237.0, [393] := 17307.0, [394] := 17004.0, [395] := 17292.0, [396] := 17209.0, [397] := 17158.0, [398] := 17100.0, [399] := 17310.0, [400] := 17254.0, [401] := 17105.0, [402] := 17157.0, [403] := 17012.0, [404] := 17310.0, [405] := 17015.0, [406] := 17152.0, [407] := 17106.0, [408] := 17258.0, [409] := 17309.0, [410] := 17043.0, [411] := 17224.0, [412] := 17119.0, [413] := 17290.0, [414] := 17003.0, [415] := 17304.0, [416] := 17239.0, [417] := 17253.0, [418] := 17021.0, [419] := 17008.0,
        [420] := 17168.0, [421] := 17201.0, [422] := 17292.0, [423] := 17004.0, [424] := 17277.0, [425] := 17082.0, [426] := 17189.0, [427] := 17073.0, [428] := 17309.0, [429] := 17279.0, [430] := 17076.0, [431] := 17122.0, [432] := 17005.0, [433] := 17308.0, [434] := 17032.0, [435] := 17247.0, [436] := 17029.0, [437] := 17311.0, [438] := 17290.0, [439] := 17067.0, [440] := 17200.0, [441] := 17173.0, [442] := 17310.0, [443] := 17029.0, [444] := 17251.0, [445] := 17088.0, [446] := 17276.0, [447] := 17009.0, [448] := 17018.0, [449] := 17210.0, [450] := 17158.0, [451] := 17260.0, [452] := 17003.0, [453] := 17299.0, [454] := 17227.0, [455] := 17129.0, [456] := 17064.0, [457] := 17285.0, [458] := 17304.0, [459] := 17075.0, [460] := 17119.0, [461] := 17024.0, [462] := 17305.0, [463] := 17031.0, [464] := 17123.0, [465] := 17127.0, [466] := 17234.0, [467] := 17305.0, [468] := 17026.0, [469] := 17242.0, [470] := 17114.0, [471] := 17277.0, [472] := 17005.0, [473] := 17306.0, [474] := 17064.0, [475] := 17285.0, [476] := 17002.0, [477] := 17073.0, [478] := 17114.0, [479] := 17246.0,
        [480] := 17305.0, [481] := 17078.0, [482] := 17177.0, [483] := 17185.0, [484] := 17306.0, [485] := 17032.0, [486] := 17236.0, [487] := 17130.0, [488] := 17310.0, [489] := 17043.0, [490] := 17140.0, [491] := 17117.0, [492] := 17292.0, [493] := 17304.0, [494] := 17034.0, [495] := 17241.0, [496] := 17251.0, [497] := 17310.0, [498] := 17008.0, [499] := 17281.0, [500] := 17124.0, [501] := 17240.0, [502] := 17033.0, [503] := 17029.0, [504] := 17250.0, [505] := 17114.0, [506] := 17216.0, [507] := 17051.0, [508] := 17299.0, [509] := 17270.0, [510] := 17093.0, [511] := 17170.0, [512] := 17204.0, [513] := 17312.0, [514] := 17013.0, [515] := 17276.0, [516] := 17186.0, [517] := 17248.0, [518] := 17029.0, [519] := 17009.0, [520] := 17289.0, [521] := 17126.0, [522] := 17239.0, [523] := 17034.0, [524] := 17310.0, [525] := 17245.0, [526] := 17120.0, [527] := 17144.0, [528] := 17305.0, [529] := 17236.0, [530] := 17127.0, [531] := 17132.0, [532] := 17036.0, [533] := 17304.0, [534] := 17003.0, [535] := 17112.0, [536] := 17147.0, [537] := 17220.0, [538] := 17291.0, [539] := 17060.0,
        [540] := 17203.0, [541] := 17160.0, [542] := 17300.0, [543] := 17003.0, [544] := 17297.0, [545] := 17158.0, [546] := 17270.0, [547] := 17012.0, [548] := 17015.0, [549] := 17217.0, [550] := 17152.0, [551] := 17256.0, [552] := 17003.0, [553] := 17301.0, [554] := 17042.0, [555] := 17140.0, [556] := 17118.0, [557] := 17247.0, [558] := 17309.0, [559] := 17007.0, [560] := 17286.0, [561] := 17195.0, [562] := 17174.0, [563] := 17085.0, [564] := 17011.0, [565] := 17310.0, [566] := 17018.0, [567] := 17161.0, [568] := 17094.0, [569] := 17267.0, [570] := 17293.0, [571] := 17053.0, [572] := 17208.0, [573] := 17152.0, [574] := 17295.0, [575] := 17000.0, [576] := 17296.0, [577] := 17228.0, [578] := 17197.0, [579] := 17056.0, [580] := 17001.0, [581] := 17303.0, [582] := 17084.0, [583] := 17197.0, [584] := 17063.0, [585] := 17299.0, [586] := 17045.0, [587] := 17143.0, [588] := 17115.0, [589] := 17293.0, [590] := 17303.0, [591] := 17036.0, [592] := 17236.0, [593] := 17126.0, [594] := 17239.0, [595] := 17032.0, [596] := 17030.0, [597] := 17242.0, [598] := 17120.0, [599] := 17226.0,
        [600] := 17042.0, [601] := 17301.0, [602] := 17003.0, [603] := 17163.0, [604] := 17092.0, [605] := 17269.0, [606] := 17192.0, [607] := 17178.0, [608] := 17081.0, [609] := 17011.0, [610] := 17310.0, [611] := 17018.0, [612] := 17098.0, [613] := 17164.0, [614] := 17199.0, [615] := 17291.0, [616] := 17004.0, [617] := 17226.0, [618] := 17140.0, [619] := 17248.0, [620] := 17028.0, [621] := 17272.0, [622] := 17171.0, [623] := 17198.0, [624] := 17065.0, [625] := 17004.0, [626] := 17305.0, [627] := 17031.0, [628] := 17119.0, [629] := 17136.0, [630] := 17231.0, [631] := 17285.0, [632] := 17069.0, [633] := 17192.0, [634] := 17176.0, [635] := 17306.0, [636] := 17005.0, [637] := 17287.0, [638] := 17071.0, [639] := 17309.0, [640] := 17008.0, [641] := 17071.0, [642] := 17196.0, [643] := 17175.0, [644] := 17275.0, [645] := 17011.0, [646] := 17290.0, [647] := 17060.0, [648] := 17164.0, [649] := 17097.0, [650] := 17303.0, [651] := 17293.0, [652] := 17053.0, [653] := 17150.0, [654] := 17042.0, [655] := 17303.0, [656] := 17004.0, [657] := 17054.0, [658] := 17214.0, [659] := 17158.0,
        [660] := 17302.0, [661] := 17006.0, [662] := 17300.0, [663] := 17048.0, [664] := 17215.0, [665] := 17052.0, [666] := 17300.0, [667] := 17268.0, [668] := 17099.0, [669] := 17163.0, [670] := 17057.0, [671] := 17296.0, [672] := 17056.0, [673] := 17151.0, [674] := 17014.0, [675] := 17312.0, [676] := 17019.0, [677] := 17093.0, [678] := 17102.0, [679] := 17262.0, [680] := 17310.0, [681] := 17012.0, [682] := 17220.0, [683] := 17107.0, [684] := 17256.0, [685] := 17021.0, [686] := 17043.0, [687] := 17223.0, [688] := 17139.0, [689] := 17294.0, [690] := 17003.0, [691] := 17301.0, [692] := 17039.0, [693] := 17136.0, [694] := 17122.0, [695] := 17240.0, [696] := 17306.0, [697] := 17031.0, [698] := 17240.0, [699] := 17141.0, [700] := 17227.0, [701] := 17038.0, [702] := 17004.0, [703] := 17294.0, [704] := 17053.0, [705] := 17156.0, [706] := 17104.0, [707] := 17300.0, [708] := 17297.0, [709] := 17049.0, [710] := 17158.0, [711] := 17215.0, [712] := 17300.0, [713] := 17005.0, [714] := 17268.0, [715] := 17164.0, [716] := 17207.0, [717] := 17063.0, [718] := 17015.0, [719] := 17274.0,
        [720] := 17086.0, [721] := 17256.0, [722] := 17023.0, [723] := 17312.0, [724] := 17012.0, [725] := 17075.0, [726] := 17190.0, [727] := 17183.0, [728] := 17308.0, [729] := 17006.0, [730] := 17284.0, [731] := 17137.0, [732] := 17283.0, [733] := 17006.0, [734] := 17027.0, [735] := 17251.0, [736] := 17111.0, [737] := 17221.0, [738] := 17046.0, [739] := 17297.0, [740] := 17297.0, [741] := 17048.0, [742] := 17219.0, [743] := 17144.0, [744] := 17247.0, [745] := 17028.0, [746] := 17307.0, [747] := 17285.0, [748] := 17067.0, [749] := 17198.0, [750] := 17034.0, [751] := 17305.0, [752] := 17004.0, [753] := 17247.0, [754] := 17025.0, [755] := 17308.0, [756] := 17006.0, [757] := 17127.0, [758] := 17129.0, [759] := 17238.0, [760] := 17308.0, [761] := 17028.0, [762] := 17245.0, [763] := 17143.0, [764] := 17308.0, [765] := 17006.0, [766] := 17065.0, [767] := 17134.0, [768] := 17286.0, [769] := 17306.0, [770] := 17030.0, [771] := 17186.0, [772] := 17185.0, [773] := 17283.0, [774] := 17007.0, [775] := 17281.0, [776] := 17187.0, [777] := 17180.0, [778] := 17082.0, [779] := 17010.0,
        [780] := 17309.0, [781] := 17017.0, [782] := 17097.0, [783] := 17160.0, [784] := 17206.0, [785] := 17310.0, [786] := 17015.0, [787] := 17267.0, [788] := 17089.0, [789] := 17256.0, [790] := 17019.0, [791] := 17310.0, [792] := 17225.0, [793] := 17143.0, [794] := 17110.0, [795] := 17021.0, [796] := 17309.0, [797] := 17010.0, [798] := 17078.0, [799] := 17186.0, [800] := 17245.0, [801] := 17026.0, [802] := 17038.0, [803] := 17137.0, [804] := 17119.0, [805] := 17243.0, [806] := 17307.0, [807] := 17006.0, [808] := 17287.0, [809] := 17202.0, [810] := 17167.0, [811] := 17091.0, [812] := 17003.0, [813] := 17293.0, [814] := 17055.0, [815] := 17211.0, [816] := 17102.0, [817] := 17262.0, [818] := 17016.0, [819] := 17106.0, [820] := 17150.0, [821] := 17219.0, [822] := 17298.0, [823] := 17003.0, [824] := 17300.0, [825] := 17227.0, [826] := 17134.0, [827] := 17060.0, [828] := 17003.0, [829] := 17304.0, [830] := 17032.0, [831] := 17172.0, [832] := 17065.0, [833] := 17307.0, [834] := 17091.0, [835] := 17205.0, [836] := 17052.0, [837] := 17289.0, [838] := 17269.0, [839] := 17080.0,
        [840] := 17178.0, [841] := 17001.0, [842] := 17299.0, [843] := 17038.0, [844] := 17228.0, [845] := 17003.0, [846] := 17295.0, [847] := 17050.0, [848] := 17213.0, [849] := 17048.0, [850] := 17300.0, [851] := 17300.0, [852] := 17047.0, [853] := 17224.0, [854] := 17116.0, [855] := 17249.0, [856] := 17026.0, [857] := 17011.0, [858] := 17234.0, [859] := 17201.0, [860] := 17064.0, [861] := 17007.0, [862] := 17309.0, [863] := 17086.0, [864] := 17197.0, [865] := 17069.0, [866] := 17312.0, [867] := 17277.0, [868] := 17084.0, [869] := 17184.0, [870] := 17006.0, [871] := 17305.0, [872] := 17041.0, [873] := 17236.0, [874] := 17126.0, [875] := 17244.0, [876] := 17030.0, [877] := 17005.0, [878] := 17286.0, [879] := 17064.0, [880] := 17230.0, [881] := 17036.0, [882] := 17305.0, [883] := 17293.0, [884] := 17112.0, [885] := 17144.0, [886] := 17044.0, [887] := 17310.0, [888] := 17021.0, [889] := 17255.0, [890] := 17088.0, [891] := 17308.0, [892] := 17027.0, [893] := 17114.0, [894] := 17083.0, [895] := 17308.0, [896] := 17287.0, [897] := 17068.0, [898] := 17204.0, [899] := 17091.0,
        [900] := 17271.0, [901] := 17016.0, [902] := 17016.0, [903] := 17270.0, [904] := 17093.0, [905] := 17170.0, [906] := 17063.0, [907] := 17291.0, [908] := 17004.0, [909] := 17030.0, [910] := 17241.0, [911] := 17121.0, [912] := 17308.0, [913] := 17007.0, [914] := 17280.0, [915] := 17188.0, [916] := 17244.0, [917] := 17027.0, [918] := 17007.0, [919] := 17284.0, [920] := 17127.0, [921] := 17128.0, [922] := 17032.0, [923] := 17304.0, [924] := 17004.0, [925] := 17059.0, [926] := 17206.0, [927] := 17280.0, [928] := 17307.0, [929] := 17026.0, [930] := 17249.0, [931] := 17144.0, [932] := 17221.0, [933] := 17039.0, [934] := 17017.0, [935] := 17250.0, [936] := 17102.0, [937] := 17148.0, [938] := 17005.0, [939] := 17305.0, [940] := 17015.0, [941] := 17227.0, [942] := 17029.0, [943] := 17298.0, [944] := 17290.0, [945] := 17102.0, [946] := 17143.0, [947] := 17043.0, [948] := 17291.0, [949] := 16998.0, [950] := 17295.0, [951] := 17223.0, [952] := 17198.0, [953] := 17051.0, [954] := 16998.0, [955] := 17299.0, [956] := 17081.0, [957] := 17193.0, [958] := 17059.0, [959] := 17296.0,
        [960] := 17219.0, [961] := 17140.0, [962] := 17114.0, [963] := 17012.0, [964] := 17264.0, [965] := 17087.0, [966] := 17103.0, [967] := 17016.0, [968] := 17309.0, [969] := 17010.0, [970] := 17141.0, [971] := 17118.0, [972] := 17244.0, [973] := 17306.0, [974] := 17005.0, [975] := 17286.0, [976] := 17200.0, [977] := 17233.0, [978] := 17034.0, [979] := 17003.0, [980] := 17246.0, [981] := 17115.0, [982] := 17135.0, [983] := 17034.0, [984] := 17301.0, [985] := 17002.0, [986] := 17054.0, [987] := 17208.0, [988] := 17219.0, [989] := 17300.0, [990] := 17002.0, [991] := 17193.0, [992] := 17081.0, [993] := 17276.0, [994] := 17010.0, [995] := 17059.0, [996] := 17204.0, [997] := 17164.0, [998] := 17095.0, [999] := 17003.0);
   NM_4303_SIGNAL_AVERAGE_WEIGHT : REAL[100];
   No_Vaild_Monomer_Barcode_Found : BOOL := 1;
   Normal_SP : REAL := 20.0;
   O5_6_PL : ALIAS FOR Local:5:O.Data.14;
   O5_9_PL : ALIAS FOR Local:5:O.Data.9;
   O7_10_BUZ : ALIAS FOR Local:7:O.Data.10;
   O7_11_BEC : ALIAS FOR Local:7:O.Data.11;
   One_Shots : DINT := 8;
   Ones4301 : DINT := 7;
   Ones4302 : DINT := 23;
   OneShots : DINT := 1073741824;
   OneShots2 : DINT;
   ons1 : BOOL := 1;
   ONS101 : BOOL := 1;
   ONS2 : BOOL;
   ONS3 : BOOL := 1;
   ons4 : BOOL := 1;
   onsB4320 : DINT;
   OnsBit : INT;
   onsT47 : DINT;
   ONSTog : DINT := 1073741860;
   OutputBit : INT;
   OutScaledMelimine : REAL;
   P_4305 : AStd_FVNR := (AutoS := 1, DiscI := 1, RuntimeS := 1079, Perm.IntlkS := 1, Perm.SafeS := 1, Perm.SafetyInhibitC := 2, Perm.IntSafDisp := 1, MiscAlm.Tmr.PRE := 10000);
   P_4305_AOI : AStd_FVNR_AOI := (AutoS := 1);
   P_S52_2_OpenC : ALIAS FOR Local:1:O.Data[12].14;
   PackTransferCompletePB : BOOL;
   PCV_4302_3 : AStd_VlvModulating := (AutoC := 1, AutoS := 1, AutoCtrlS := 1, Perm.IntlkS := 1, Perm.SafeS := 1, AutoCtrlC := 1, AutoPosC[1] := 100.0, Scaling.RawMaxS := 10000.0, Scaling.EngMaxS := 100.0);
   PCV_4302_3_AOI : AStd_VlVModulating_AOI := (cfgEUMax := 100.0, cfgRawMax := 10000.0, AutoS := 1);
   Phase_AlarmHorn : BOOL;
   PhaseHornONS : DINT;
   PIC_4302_3 : AStd_PIDInterface := (AutoS := 1, AutoCtrlC := 1, AutoCtrlS := 1, EnableS := 1, ManOut := 100.0, SPC := 15.0, PGainC := 7.5, IGainC := 0.1, PGainS := 7.5, IGainS := 0.1, SPS := 15.0, PVS := 17.549, CVS := 100.0, Perm.IntlkS := 1, Perm.SafeS := 1);
   PIC_4302_3_AOI : AStd_PIDInterface_AOI := (SP := 15.0, PV := 17.556, CV := 100.0, cfgPVMaxEU := 60.0);
   PIC_4302_3_Mode : SINT := 1;
   PIC_4302_3_PID : PID_ENHANCED := (PV := 17.555, PVEUMax := 60.0, SPProg := 15.0, SPOper := 15.0, SPHLimit := 60.0, RatioProg := 1.0, RatioOper := 1.0, RatioHLimit := 1.0, RatioLLimit := 1.0, CVProg := 100.0, CVOper := 100.0, CVEUMax := 100.0, CVHLimit := 100.0, ControlAction := 1, DependIndepend := 1, PGain := 7.5, IGain := 0.1, DevHHLimit := 5.0, ProgProgReq := 1, ProgAutoReq := 1, RTSTime := 1, CVEU := 100.0, CV := 100.0, CVHAlarm := 1, SP := 15.0, SPPercent := 25.0, PVPercent := 29.248333, E := 2.5489998, EPercent := 4.248333, InitPrimary := 1, WindupLOut := 1, Ratio := 1.0, ProgOper := 1, Auto := 1, DeltaT := 0.1);
   PIC_4302_3_Setpoint : REAL := 15.0;
   PID_T4301C : PID := (CTL := 304124416, PVT := 1, CA := 1, NOBC := 1, INI := 1, OLH := 1, DVPA := 1, SP := 85.0, KP := 325.0, KI := 0.02, MAXS := 4095.0, SO := 100.0, MAXO := 100.0, UPD := 1.0, PV := 99.0, ERR := 14.0, PVH := 1000.0, MAXI := 4095.0, MAXCV := 10000.0, MAXTIE := 100.0, DATA[1] := 38.68132, DATA[2] := 99.0, DATA[3] := 14.0, DATA[4] := 85.0, DATA[5] := 0.024420025, DATA[6] := 1.0, DATA[7] := 16.0, DATA[8] := 325.0, DATA[9] := 0.02, DATA[11] := 325.0, DATA[12] := 0.02, DATA[15] := 100.0, DATA[16] := 1.0);
   PID_T4301Com : PID;
   PID_T4301H : PID := (CTL := 270570112, PVT := 1, NOBC := 1, INI := 1, OLH := 1, DVPA := 1, PVHA := 1, SP := 150.0, KP := 8.0, KI := 0.2, MAXS := 4095.0, SO := 100.0, MAXO := 50.0, UPD := 1.0, PV := 146.0, ERR := 4.0, MAXI := 4095.0, MAXCV := 10000.0, MAXTIE := 100.0, DATA[1] := -57.045177, DATA[2] := 146.0, DATA[3] := 4.0, DATA[4] := 150.0, DATA[5] := 0.024420025, DATA[6] := 1.0, DATA[7] := 16.0, DATA[8] := 8.0, DATA[9] := 0.2, DATA[11] := 8.0, DATA[12] := 0.2, DATA[15] := 100.0, DATA[16] := 1.0);
   PID_T4302C : PID := (CTL := -1843354624, EN := 1, PVT := 1, CA := 1, NOBC := 1, INI := 1, OLL := 1, DVNA := 1, SP := 180.0, KP := 150.0, KI := 0.01, MAXS := 4095.0, MAXO := 100.0, UPD := 0.6, PV := 65.0, ERR := -115.0, PVH := 1000.0, MAXI := 4095.0, MAXCV := 10000.0, MAXTIE := 100.0, DATA[0] := 3.6631439, DATA[1] := 25.396826, DATA[2] := 65.0, DATA[3] := -115.0, DATA[4] := 180.0, DATA[5] := 0.024420025, DATA[6] := 1.0, DATA[7] := 9.6, DATA[8] := 150.0, DATA[9] := 0.01, DATA[11] := 150.0, DATA[12] := 0.01, DATA[15] := 100.0, DATA[16] := 1.0);
   PID_T4302H : PID := (CTL := 270537344, PVT := 1, NOBC := 1, OLH := 1, DVPA := 1, PVHA := 1, SP := 150.0, KP := 8.0, KI := 0.2, MAXS := 4095.0, SO := 50.0, MAXO := 50.0, UPD := 1.0, PV := 174.0, ERR := 106.0, MAXI := 4095.0, MAXCV := 10000.0, MAXTIE := 100.0, DATA[1] := -67.98535, DATA[2] := 174.0, DATA[3] := 106.0, DATA[4] := 280.0, DATA[5] := 0.024420025, DATA[6] := 1.0, DATA[7] := 16.0, DATA[8] := 8.0, DATA[9] := 0.2, DATA[11] := 8.0, DATA[12] := 0.2, DATA[15] := 100.0, DATA[16] := 1.0);
   PIDE_TCV_S47_1 : PID_ENHANCED := (PV := 68.1075, PVEUMax := 200.0, SPProg := 32.8275, SPOper := 50.0, SPHLimit := 150.0, SPLLimit := 50.0, RatioProg := 1.0, RatioOper := 1.0, RatioHLimit := 1.0, RatioLLimit := 1.0, CVEUMax := 100.0, CVHLimit := 100.0, PGain := 10.0, IGain := 1.0, PVEDerivative := 1, ProgOverrideReq := 1, RTSTime := 1, SP := 50.0, SPPercent := 25.0, PVPercent := 34.05375, E := -18.107498, EPercent := -9.053749, InitPrimary := 1, Ratio := 1.0, Override := 1, DeltaT := 0.1, Status1 := 16#0000_0021, InstructFault := 1, SPProgInv := 1);
   PIDE_TCV_S47_1_AutoSP : REAL := 32.8275;
   PIDTMRCOOL : TIMER := (PRE := 5000, ACC := 5000, EN := 1, DN := 1);
   PIDTMRCOOL2 : TIMER := (PRE := 5000, ACC := 5001, EN := 1, DN := 1);
   PIT_4302_2 : AStd_AnalogInput := (Raw := -12450.0, Scaled := 17.55, Scaling.RawMinS := -30000.0, Scaling.RawMaxS := 30000.0, Scaling.EngMaxS := 60.0, LowLow.LimitC := 10.0, LowLow.Tmr.PRE := 1000, LowLow.Disabled := 1, Low.LimitC := 20.0, Low.Tmr.PRE := 1000, Low.Disabled := 1, High.LimitC := 280.0, High.Tmr.PRE := 1000, High.Disabled := 1, HighHigh.LimitC := 290.0, HighHigh.Tmr.PRE := 1000, HighHigh.Disabled := 1, Fault.LimitC := -31000.0, Fault.LimitOffSetC := 1000.0, Fault.Tmr.PRE := 1000, FaultReset := 500.0);
   PIT_4302_2_AOI : AStd_AI_AOI := (InputRaw_I := -12445.0, cfgRawMin := -30000.0, cfgRawMax := 30000.0, cfgEUMax := 60.0, Scaled := 17.555);
   PIT_4302_2_Holding : DINT := -12457;
   PIT_4302_2_Samples : DINT := 100;
   PIT_4302_2_sim_Val : DINT := 25;
   PIT_4302_2_Simulation : BOOL := 1;
   PLCStatus : AStd_PLCStatus := (MinorFaultBits := 24, PLCScanTime := 17.855, PLCScanTimeMin := 0.00029758332, DateTime.CurrentYear := 2001, DateTime.CurrentMonth := 6, DateTime.CurrentDay := 2, DateTime.CurrentHour := 17, DateTime.CurrentMinute := 43, DateTime.CurrentSecond := 6, DateTime.DateTimeBuild := '62200117436', DateTime.TemporaryString := '6', DateTime.DateTimeBuffer[0] := 2001, DateTime.DateTimeBuffer[1] := 6, DateTime.DateTimeBuffer[2] := 2, DateTime.DateTimeBuffer[3] := 17, DateTime.DateTimeBuffer[4] := 43, DateTime.DateTimeBuffer[5] := 6, DateTime.DateTimeBuffer[6] := 480979, DateTime.CurrentDateTime := '62200117436', PLCPowerUp.LatchA := 1);
   PowerLimit : REAL;
   PS_AirMakeup : ALIAS FOR Local:1:I.Data[33].3;
   PulseBit : INT;
   PulseToLbFactor : REAL := 5.0;
   Pump_Enable_TMR : TIMER := (PRE := 300000);
   PUMP_P_4305_AUX : ALIAS FOR Local:1:I.Data[1].7;
   PUMP_P_4305_RUN : ALIAS FOR Local:1:O.Data[0].7;
   Pump_Running_Monmomer_Fill : BOOL;
   Pv_Disp_Alarm_Val : DINT := 103;
   Pv_Inx_Alarm_Val : DINT := 11;
   ReffVfd : VFD;
   RESET_INTERLOCK_TEST_BUTTON : BOOL;
   resetTimer : BOOL;
   RG_T51 : REAL := 48707.535;
   RG_T51_AI_Holding : REAL := 14390.579;
   RG_T51_AI_Raw : INT := 14391;
   RG_T51_AI_Samples : DINT := 1000;
   RG_T51_FILL : REAL;
   RG_T51_Holding1 : REAL := 14390.94;
   RG_T51_Min_Tank_Value : INT := 1500;
   RG_T51_OffSet : REAL := 4000.0;
   RG_T51_REMAINDER : REAL;
   RG_T51_Sf : REAL := 4.6875;
   RG_T51_Warn : REAL := 71250.0;
   RG_T52 : REAL := 100799.766;
   RG_T52_AI_Holding : REAL := 20999.744;
   RG_T52_AI_Raw : INT := 21000;
   RG_T52_AI_Samples : DINT := 100;
   RG_T52_FULL : REAL;
   RG_T52_Holding1 : REAL := 20999.477;
   RG_T52_Min_Tank_Value : INT := 1;
   RG_T52_OffSet : REAL := 6075.0;
   RG_T52_REMAINDER : REAL;
   RG_T52_Sf : REAL := 6.75399;
   RG_T52_Warn : REAL := 104000.0;
   RG_T53 : REAL := 59755.336;
   RG_T53_AI_Holding : REAL := 12847.621;
   RG_T53_AI_Raw : INT := 12854;
   RG_T53_AI_Samples : DINT := 100;
   RG_T53_FULL : REAL;
   RG_T53_Holding1 : REAL := 12847.412;
   RG_T53_Min_Tank_Value : INT := 15000;
   RG_T53_OffSet : REAL := 4000.0;
   RG_T53_REMAINDER : REAL;
   RG_T53_Sf : REAL := 6.75399;
   RG_T53_Warn : REAL := 104000.0;
   RM_High_Timer : TIMER := (PRE := 1500);
   RM_Pump_P51_Aux : ALIAS FOR Local:1:I.Data[33].2;
   RM_Pump_P51_Run : ALIAS FOR Local:1:O.Data[13].0;
   RM_Pump_P51_Run_PB : ALIAS FOR Local:1:I.Data[40].0;
   RM_Pump_P51_Run_PB_2 : ALIAS FOR Local:1:I.Data[40].2;
   RM_Pump_P51_RunA : ALIAS FOR Local:1:O.Data[23].0;
   RM_Pump_P51_Stop_PB : ALIAS FOR Local:1:I.Data[40].1;
   RM_Pump_T51_Run_Lamp : ALIAS FOR Local:1:O.Data[12].2;
   RM_Pump_T51_Run_Lamp2 : ALIAS FOR Local:1:O.Data[0].20;
   RM_Pump_T51_Run_LampA : ALIAS FOR Local:1:O.Data[22].2;
   RM_Tank_T51_Fill_Closed : ALIAS FOR Local:1:O.Data[12].10;
   RM_Tank_T51_Fill_ClosedA : ALIAS FOR Local:1:O.Data[22].10;
   RM_Tank_T51_Level_Lamp : ALIAS FOR Local:1:O.Data[12].5;
   RM_Tank_T51_Level_LampA : ALIAS FOR Local:1:O.Data[22].5;
   RM_To_W2 : ALIAS FOR Local:1:I.Data[1].20;
   RM_To_W4 : ALIAS FOR Local:1:I.Data[1].21;
   RO_END : TIMER := (PRE := 5000);
   RO_HE4305_PhaseROHotWaterDrop : AStd_PLI := (IdleS := 1, CurrentStateCodeS := 1, StepNo := 1, StepBit := 2, PreventStartInhibitC := 31, AlarmInhibitC := 31);
   RO_HE4305_PhaseROHotWaterDrop_AOI : AStd_PLI_AOI := (StepNo := 1, cfgAutoReset := 1);
   RO_HE4305_PhaseROWaterAddition : AStd_PLI := (IdleS := 1, CurrentStateCodeS := 1, PreventStartS := 64, AlarmS := 64, StepNo := 1, StepBit := 2, RealParameters[0] := 59.0, RealParameters[1] := 49.0, RealParameters[4] := 2.0, RealParameters[5] := 65.0, RealParameters[6] := 59.0, RealParameters[7] := 1.0, RealParameters[8] := 10.0, RealParameters[9] := 49.0, RealParameters[17] := 4.0, RealParameters[18] := 994.881, RealParameters[19] := 51.007023, PreventStartInhibitC := 511, AlarmInhibitC := 511, IntSafDisp := 64, InterlockTimers.Timers[3].PRE := 3000, InterlockTimers.Timers[3].ACC := 3004, InterlockTimers.Timers[3].EN := 1, InterlockTimers.Timers[3].DN := 1);
   RO_HE4305_PhaseROWaterAddition_AOI : AStd_PLI_AOI := (PreventStartS := 1, AlmS := 1, StepNo := 1, cfgAutoReset := 1);
   Ro_MaxFeedRate : REAL := 124.0;
   RO_PERCENT_VALVE : REAL := 29.0;
   RO_Preheat_Temp : DINT := 50;
   ROC_SP : REAL := 1.08;
   ROC_SP_10min : REAL := 10.8;
   ROWaterAdd_StepComplete : BOOL[32];
   RTA_Input_Coils : SINT[50];
   RTA_Input_Floats : REAL[100] := ([1] := 10714.0, [2] := 10715.0);
   RTA_Status_Coils : SINT[50];
   S4352_Phase_Circulation : AStd_PLI := (IdleS := 1, CurrentStateCodeS := 1, PreventStartS := 2, AlarmS := 2, StepNo := 1, StepBit := 2, RealParameters[0] := 60.0, DINTParameters[0] := 10, PreventStartInhibitC := 7, AlarmInhibitC := 3, IntSafDisp := 2);
   S4352_Phase_Circulation_AOI : AStd_PLI_AOI := (PreventStartS := 1, AlmS := 1, StepNo := 1, cfgAutoReset := 1);
   S4352_Phase_Packaging_Transfer : AStd_PLI := (IdleS := 1, CurrentStateCodeS := 1, PreventStartS := 2, AlarmS := 2, StepNo := 1, StepBit := 2, PreventStartInhibitC := 7, AlarmInhibitC := 3, IntSafDisp := 2);
   S4352_Phase_Packaging_Transfer_AOI : AStd_PLI_AOI := (PreventStartS := 1, AlmS := 1, StepNo := 1, cfgAutoReset := 1);
   S4352_Phase_TT_Transfer : AStd_PLI := (IdleS := 1, CurrentStateCodeS := 1, PreventStartS := 2, AlarmS := 2, StepNo := 1, StepBit := 2, RealParameters[0] := 44000.0, PreventStartInhibitC := 7, AlarmInhibitC := 3, IntSafDisp := 2);
   S4352_Phase_TT_Transfer_AOI : AStd_PLI_AOI := (PreventStartS := 1, AlmS := 1, StepNo := 1, cfgAutoReset := 1);
   S4352_PhaseTransfer : AStd_PLI; {access Read Only}
   S4352_TransferStarted : BOOL;
   S47_HighHighLevel : BOOL;
   S47_HighHighLevelMessage : BOOL;
   S47_HighLevel : BOOL := 1;
   S47_LastTrasferredLb : REAL := 5.0;
   S47_OkToRun : BOOL;
   S47_PumpAutoCommand : BOOL;
   S47_PumpIsRunning : BOOL;
   S47_PumpManCommand : BOOL;
   S47_PumpManStartPB : BOOL;
   S47_PumpManStopPB : BOOL;
   S47_Selected : BOOL;
   S47_SelectPB : BOOL;
   S47_Toggle : AOI_Toggle := (QNot := 1);
   S47_transfer_amount : REAL;
   S47_TransferLimit : REAL := 44500.0;
   S47_transferLimitMessage : BOOL;
   S47_TransferSetpoint : REAL;
   S47_TransferStarted : BOOL;
   S47_TransferStartPB : BOOL;
   S47_TransferStopPB : BOOL;
   S52_Circulation_StopPB : BOOL;
   S52_Circulation_Timer : TIMER;
   S52_Circulation_Timer_Mins : DINT;
   S52CirculationRemMins : REAL;
   S52TotalizerBypassPB : BOOL;
   S52TransferCompletePB : BOOL;
   SaveBarcode : BOOL;
   ScreenDisplayBarcode : STRING;
   Shortstop_Activate : BOOL;
   Shortstop_Temperature : REAL;
   Shortstop_Timer : TIMER[10];
   Shortstop_Timer_1 : REAL := 10.0;
   Shortstop_Timer_2 : REAL := 45.0;
   SIL2_from_Dispersion : DINT;
   SIL2_from_Dispersion_Analog : REAL[24];
   SIL2_from_Dispersion_Analog_xxx : DINT;
   SIL2_to_Dispersion : DINT := 41349;
   SIL2_to_Dispersion_Analog : REAL[24];
   Source : DINT;
   Source_Selection : BOOL := 1;
   SP : REAL := 112.999985;
   SPARE_I10_00 : REAL;
   SPARE_I10_01 : REAL;
   SPARE_I10_02 : REAL;
   SPARE_I10_03 : REAL;
   SPARE_I10_04 : REAL;
   SPARE_I10_05 : REAL;
   SPARE_I204 : ALIAS FOR Local:2:I.Data.4;
   SPARE_I205 : ALIAS FOR Local:2:I.Data.5;
   SPARE_I301 : ALIAS FOR Local:3:I.Data.1;
   SPARE_I302 : ALIAS FOR Local:3:I.Data.2;
   SPARE_I303 : ALIAS FOR Local:3:I.Data.3;
   SPARE_I304 : ALIAS FOR Local:3:I.Data.4;
   SPARE_I305 : ALIAS FOR Local:3:I.Data.5;
   SPARE_I306 : ALIAS FOR Local:3:I.Data.6;
   SPARE_I307 : ALIAS FOR Local:3:I.Data.7;
   SPARE_I308 : ALIAS FOR Local:3:I.Data.8;
   SPARE_I309 : ALIAS FOR Local:3:I.Data.9;
   SPARE_I310 : ALIAS FOR Local:3:I.Data.10;
   SPARE_I311 : ALIAS FOR Local:3:I.Data.11;
   SPARE_I312 : ALIAS FOR Local:3:I.Data.12;
   SPARE_I313 : ALIAS FOR Local:3:I.Data.13;
   SPARE_I314 : ALIAS FOR Local:3:I.Data.14;
   SPARE_I315 : ALIAS FOR Local:3:I.Data.14;
   SPARE_I400 : ALIAS FOR Local:4:I.Data.0;
   SPARE_I401 : ALIAS FOR Local:4:I.Data.1;
   SPARE_I402 : ALIAS FOR Local:4:I.Data.2;
   SPARE_I403 : ALIAS FOR Local:4:I.Data.3;
   SPARE_I404 : ALIAS FOR Local:4:I.Data.4;
   SPARE_I405 : ALIAS FOR Local:4:I.Data.5;
   SPARE_I406 : ALIAS FOR Local:4:I.Data.6;
   SPARE_I407 : ALIAS FOR Local:4:I.Data.7;
   SPARE_I408 : ALIAS FOR Local:4:I.Data.8;
   SPARE_I409 : ALIAS FOR Local:4:I.Data.9;
   SPARE_I410 : ALIAS FOR Local:4:I.Data.10;
   SPARE_I411 : ALIAS FOR Local:4:I.Data.11;
   SPARE_I412 : ALIAS FOR Local:4:I.Data.12;
   SPARE_I413 : ALIAS FOR Local:4:I.Data.13;
   SPARE_I414 : ALIAS FOR Local:4:I.Data.14;
   SPARE_I415 : ALIAS FOR Local:4:I.Data.15;
   SPARE_I_1_1_18 : ALIAS FOR Local:1:I.Data[1].18;
   SPARE_I_1_1_19 : ALIAS FOR Local:1:I.Data[1].19;
   SPARE_I_1_1_20 : ALIAS FOR Local:1:I.Data[1].20;
   SPARE_I_1_1_21 : ALIAS FOR Local:1:I.Data[1].21;
   SPARE_I_1_1_22 : ALIAS FOR Local:1:I.Data[1].22;
   SPARE_I_1_1_23 : ALIAS FOR Local:1:I.Data[1].23;
   SPARE_I_1_4_4 : ALIAS FOR Local:1:I.Data[4].4;
   SPARE_I_1_4_5 : ALIAS FOR Local:1:I.Data[4].5;
   SPARE_I_1_4_6 : ALIAS FOR Local:1:I.Data[4].6;
   SPARE_I_1_4_7 : ALIAS FOR Local:1:I.Data[4].7;
   SPARE_I_1_77 : REAL;
   SPARE_I_1_78 : REAL;
   SPARE_I_1_79 : REAL;
   SPARE_I_1_80 : REAL;
   SPARE_I_1_81 : REAL;
   SPARE_I_1_85 : REAL;
   SPARE_I_1_86 : REAL;
   SPARE_I_1_87 : REAL;
   SPARE_I_1_88 : REAL;
   SPARE_I_1_89 : REAL;
   SPARE_I_1_90 : REAL;
   SPARE_I_1_91 : REAL;
   SPARE_I_2_4 : REAL;
   SPARE_I_2_6 : REAL;
   SPARE_I_2_7 : REAL;
   SPARE_O502 : ALIAS FOR Local:5:O.Data.2;
   SPARE_O510 : ALIAS FOR Local:5:O.Data.10;
   SPARE_O512 : ALIAS FOR Local:5:O.Data.12;
   SPARE_O513 : ALIAS FOR Local:5:O.Data.13;
   SPARE_O514 : ALIAS FOR Local:5:O.Data.14;
   SPARE_O515 : ALIAS FOR Local:5:O.Data.15;
   SPARE_O600 : ALIAS FOR Local:6:O.Data.0;
   SPARE_O601 : ALIAS FOR Local:6:O.Data.1;
   SPARE_O602 : ALIAS FOR Local:6:O.Data.2;
   SPARE_O603 : ALIAS FOR Local:6:O.Data.3;
   SPARE_O604 : ALIAS FOR Local:6:O.Data.4;
   SPARE_O605 : ALIAS FOR Local:6:O.Data.5;
   SPARE_O606 : ALIAS FOR Local:6:O.Data.6;
   SPARE_O607 : ALIAS FOR Local:6:O.Data.7;
   SPARE_O609 : ALIAS FOR Local:6:O.Data.9;
   SPARE_O610 : ALIAS FOR Local:6:O.Data.10;
   SPARE_O611 : ALIAS FOR Local:6:O.Data.11;
   SPARE_O612 : ALIAS FOR Local:6:O.Data.12;
   SPARE_O613 : ALIAS FOR Local:6:O.Data.13;
   SPARE_O614 : ALIAS FOR Local:6:O.Data.14;
   SPARE_O615 : ALIAS FOR Local:6:O.Data.15;
   SPARE_O700 : ALIAS FOR Local:7:O.Data.0;
   SPARE_O701 : ALIAS FOR Local:7:O.Data.1;
   SPARE_O702 : ALIAS FOR Local:7:O.Data.2;
   SPARE_O703 : ALIAS FOR Local:7:O.Data.3;
   SPARE_O704 : ALIAS FOR Local:7:O.Data.4;
   SPARE_O705 : ALIAS FOR Local:7:O.Data.5;
   SPARE_O706 : ALIAS FOR Local:7:O.Data.6;
   SPARE_O707 : ALIAS FOR Local:7:O.Data.7;
   SPARE_O714 : ALIAS FOR Local:7:O.Data.14;
   SPARE_O715 : ALIAS FOR Local:7:O.Data.15;
   SPARE_O_13_1 : ALIAS FOR Local:13:O.Ch1Data;
   SPARE_O_1_0_19 : ALIAS FOR Local:1:O.Data[0].19;
   SPARE_O_1_0_20 : ALIAS FOR Local:1:O.Data[0].20;
   SPARE_O_1_0_21 : ALIAS FOR Local:1:O.Data[0].21;
   SPARE_O_1_0_22 : ALIAS FOR Local:1:O.Data[0].22;
   SPARE_O_1_0_23 : ALIAS FOR Local:1:O.Data[0].23;
   SPARE_O_1_1_10 : ALIAS FOR Local:1:O.Data[1].10;
   SPARE_O_1_1_11 : ALIAS FOR Local:1:O.Data[1].11;
   SPARE_O_1_1_12 : ALIAS FOR Local:1:O.Data[1].12;
   SPARE_O_1_1_13 : ALIAS FOR Local:1:O.Data[1].13;
   SPARE_O_1_1_14 : ALIAS FOR Local:1:O.Data[1].14;
   SPARE_O_1_1_2 : ALIAS FOR Local:1:O.Data[1].2;
   SPARE_O_1_1_3 : ALIAS FOR Local:1:O.Data[1].3;
   SPARE_O_1_1_4 : ALIAS FOR Local:1:O.Data[1].4;
   SPARE_O_1_1_5 : ALIAS FOR Local:1:O.Data[1].5;
   SPARE_O_1_1_6 : ALIAS FOR Local:1:O.Data[1].6;
   SPARE_O_1_1_7 : ALIAS FOR Local:1:O.Data[1].7;
   SPARE_O_1_1_8 : ALIAS FOR Local:1:O.Data[1].8;
   SRT_PB_BL_4310 : ALIAS FOR Local:2:I.Data.13;
   SRT_PB_P_4310 : ALIAS FOR Local:2:I.Data.15;
   ST_K400_1 : REAL := 86.07751;
   ST_K400_1_HIGH : REAL := 100.0;
   ST_K400_1_LOW : REAL := 74.0;
   ST_K400_1_Timer : TIMER[6] := ([0].PRE := 1000, [1].PRE := 1000);
   ST_K400_SAFETY : BOOL;
   Start_B4320_Transfer_PB : BOOL;
   Start_Melamine_Transfer_PB : BOOL;
   Start_T47_Transfer_PB : BOOL;
   StorageBit : INT;
   STP_PB_BL_4310 : ALIAS FOR Local:2:I.Data.14;
   STP_PB_P_4310 : ALIAS FOR Local:3:I.Data.0;
   SV_4302_1 : AStd_VlvOC := (CloseO := 1, ClosedI := 1, CycleCountS := 284, Perm.IntlkS := 1, Perm.SafeS := 1, MiscAlm.Tmr.PRE := 30000);
   SV_4302_1_AOI : AStd_VlvOC_AOI := (Close_O := 1);
   SV_4302_1_ICls : BOOL;
   SV_4302_1_IOls : BOOL;
   SV_4302_1_OClose : BOOL := 1;
   SV_4303_01 : ALIAS FOR Local:5:O.Data.8;
   SV_4303_02 : ALIAS FOR Local:7:O.Data.9;
   SV_4303_02_ZSC : BOOL := 1;
   SV_4303_02_ZSO : BOOL;
   SV_4303_03 : BOOL;
   SV_4303_03_Enable_PB : BOOL;
   SV_4303_04 : BOOL;
   SV_4303_04_Enable_PB : BOOL;
   SV_4304 : ALIAS FOR Local:5:O.Data.11;
   SV_4304_02 : BOOL;
   SV_4304_02_Enable_PB : BOOL;
   SV_4304_03 : BOOL;
   SV_4304_03_Enable_PB : BOOL;
   SV_4306_1 : AStd_VlvOC := (AutoS := 1, CloseO := 1, ClosedI := 1, CycleCountS := 2339, Perm.IntlkS := 1, Perm.SafeS := 1, MiscAlm.Tmr.PRE := 30000);
   SV_4306_1_AOI : AStd_VlvOC_AOI := (AutoS := 1, Close_O := 1);
   SV_4307_1 : AStd_VlvOC := (AutoS := 1, CloseO := 1, ClosedI := 1, CycleCountS := 1011, Perm.IntlkS := 1, Perm.SafeS := 1, MiscAlm.Tmr.PRE := 30000);
   SV_4307_1_AOI : AStd_VlvOC_AOI := (AutoS := 1, Close_O := 1);
   SV_4310 : ALIAS FOR Local:5:O.Data.5;
   SV_S52_2 : AStd_VlvOC := (CloseO := 1, ClosedI := 1, CycleCountS := 79, Perm.IntlkS := 1, Perm.SafeS := 1, MiscAlm.Tmr.PRE := 30000);
   SV_S52_2_AOI : AStd_VlvOC_AOI := (Close_O := 1); {access Read Only}
   SV_S52_2_OpenC : ALIAS FOR Local:1:O.Data[12].14;
   T0110_PhaseTimedAgitate : AStd_PLI := (IdleS := 1, CurrentStateCodeS := 1, StepNo := 1, StepBit := 2, UnitProc_PhaseID := 1111);
